// TIA Portal V20 export
FUNCTION_BLOCK "LER_IRCheck_BT5525"   // FB19, LAD
// stored: Access Published, MemoryReserve 100, SetENOAutomatically false
   VAR_INPUT
      enable : Bool;
      enableManualCmds : Bool;
      dryRunCmds : Bool;
   END_VAR
   VAR_OUTPUT
      error : Bool;
      status : Word;
   END_VAR
   VAR_IN_OUT
      controlNode : "LER_typeHipotControlNodes";
      configuration : "LER_typeHipotConfiguration";
      moduleInterface : "LER_typeHipotInterface";
   END_VAR
   VAR
      instSendP2P_type1 { ExternalAccessible := 'False'; ExternalVisible := 'False'; ExternalWritable := 'False'} : Send_P2P;
      instSendP2P_contact { S7_SetPoint := 'True'} : Send_P2P;
      instSendP2P_bddCount { S7_SetPoint := 'True'} : Send_P2P;
      instSendP2P_bddResult { S7_SetPoint := 'True'} : Send_P2P;
      instSendP2P_voltageCmd { S7_SetPoint := 'True'} : Send_P2P;
      instSendP2P_voltageCheck { S7_SetPoint := 'True'} : Send_P2P;
      instSendP2P_timerCmd { S7_SetPoint := 'True'} : Send_P2P;
      instSendP2P_timerCheck { S7_SetPoint := 'True'} : Send_P2P;
      instSendP2P_contactCmd { S7_SetPoint := 'True'} : Send_P2P;
      instSendP2P_contactCheck { S7_SetPoint := 'True'} : Send_P2P;
      instSendP2P_comparatorCmd { S7_SetPoint := 'True'} : Send_P2P;
      instSendP2P_comparatorCheck { S7_SetPoint := 'True'} : Send_P2P;
      instSendP2P_BDD_CCV_cmd { S7_SetPoint := 'True'} : Send_P2P;
      instSendP2P_BDD_CCV_check { S7_SetPoint := 'True'} : Send_P2P;
      instSendP2P_BDD_CVV_cmd { S7_SetPoint := 'True'} : Send_P2P;
      instSendP2P_BDD_CVV_check { S7_SetPoint := 'True'} : Send_P2P;
      instSendP2P_BDD_CVI_cmd { S7_SetPoint := 'True'} : Send_P2P;
      instSendP2P_BDD_CVI_check { S7_SetPoint := 'True'} : Send_P2P;
      instReceiveP2P_type1 { ExternalAccessible := 'False'; ExternalVisible := 'False'; ExternalWritable := 'False'} : Receive_P2P;
      instReceiveP2P_contact { ExternalAccessible := 'False'; ExternalVisible := 'False'; ExternalWritable := 'False'} : Receive_P2P;
      instReceiveP2P_bddCount { ExternalAccessible := 'False'; ExternalVisible := 'False'; ExternalWritable := 'False'} : Receive_P2P;
      instReceiveP2P_bddResult { S7_SetPoint := 'True'} : Receive_P2P;
      instReceiveP2P_voltageCheck { S7_SetPoint := 'True'} : Receive_P2P;
      instReceiveP2P_timerCheck { S7_SetPoint := 'True'} : Receive_P2P;
      instReceiveP2P_contactCheck { S7_SetPoint := 'True'} : Receive_P2P;
      instReceiveP2P_comparatorCheck { S7_SetPoint := 'True'} : Receive_P2P;
      instReceiveP2P_BDD_CCV_check { S7_SetPoint := 'True'} : Receive_P2P;
      instReceiveP2P_BDD_CVV_check { S7_SetPoint := 'True'} : Receive_P2P;
      instReceiveP2P_BDD_CVI_check { S7_SetPoint := 'True'} : Receive_P2P;
      instReceiveReset_type1 { ExternalAccessible := 'False'; ExternalVisible := 'False'; ExternalWritable := 'False'} : Receive_Reset;
      instReceiveReset_contact { S7_SetPoint := 'True'} : Receive_Reset;
      instReceiveReset_bddCount { S7_SetPoint := 'True'} : Receive_Reset;
      instReceiveReset_bddResult { S7_SetPoint := 'True'} : Receive_Reset;
      instReceiveReset_voltageCheck { S7_SetPoint := 'True'} : Receive_Reset;
      instReceiveReset_timerCheck { S7_SetPoint := 'True'} : Receive_Reset;
      instReceiveReset_contactCheck { S7_SetPoint := 'True'} : Receive_Reset;
      instReceiveReset_comparatorCheck { S7_SetPoint := 'True'} : Receive_Reset;
      instReceiveReset_BDD_CCV_check { S7_SetPoint := 'True'} : Receive_Reset;
      instReceiveReset_BDD_CVV_check { S7_SetPoint := 'True'} : Receive_Reset;
      instReceiveReset_BDD_CVI_check { S7_SetPoint := 'True'} : Receive_Reset;
      LER_IRCheck_Calculate_Voltage { S7_SetPoint := 'True'} : "LER_IRCheck_Calculate";
      LER_IRCheck_Calculate_Timer { S7_SetPoint := 'True'} : "LER_IRCheck_Calculate";
      LER_IRCheck_Calculate_ContactCheckLimit { S7_SetPoint := 'True'} : "LER_IRCheck_Calculate";
      LER_IRCheck_Calculate_CompUpperLimit { S7_SetPoint := 'True'} : "LER_IRCheck_Calculate";
      LER_IRCheck_Calculate_CompLowerLimit { S7_SetPoint := 'True'} : "LER_IRCheck_Calculate";
      LER_IRCheck_Calculate_CompLowerLimit_1 { S7_SetPoint := 'True'} : "LER_IRCheck_Calculate";
      LER_IRCheck_Calculate_CompLowerLimit_2 { S7_SetPoint := 'True'} : "LER_IRCheck_Calculate";
      LER_IRCheck_Calculate_CompLowerLimit_3 { S7_SetPoint := 'True'} : "LER_IRCheck_Calculate";
      LER_IRCheck_Calculate_CompLowerLimit_4 { S7_SetPoint := 'True'} : "LER_IRCheck_Calculate";
      LER_IRCheck_Calculate_CompLowerLimit_5 { S7_SetPoint := 'True'} : "LER_IRCheck_Calculate";
      LER_IRCheck_Calculate_BDD_CCV_Set { S7_SetPoint := 'True'} : "LER_IRCheck_Calculate";
      LER_IRCheck_Calculate_BDD_CVV_Set { S7_SetPoint := 'True'} : "LER_IRCheck_Calculate";
      LER_IRCheck_Calculate_BDD_CVI_Set { S7_SetPoint := 'True'} : "LER_IRCheck_Calculate";
      instTON_type1 { S7_SetPoint := 'True'} : Array[0..4] of TON_TIME;
      instTON_contact { S7_SetPoint := 'True'} : Array[0..4] of TON_TIME;
      instTON_bddCount { S7_SetPoint := 'True'} : Array[0..4] of TON_TIME;
      instTON_bddResult { S7_SetPoint := 'True'} : Array[0..4] of TON_TIME;
      instTON_voltage { S7_SetPoint := 'True'} : Array[0..4] of TON_TIME;
      instTON_delayTest { S7_SetPoint := 'True'} : Array[0..4] of TON_TIME;
      statSendP2PLength_type1 { ExternalAccessible := 'False'; ExternalVisible := 'False'; ExternalWritable := 'False'} : UInt;
      statSendP2PLength_contact { ExternalAccessible := 'False'; ExternalVisible := 'False'; ExternalWritable := 'False'} : UInt;
      statSendP2PLength_bddCount { ExternalAccessible := 'False'; ExternalVisible := 'False'; ExternalWritable := 'False'} : UInt;
      statSendP2PLength_bddResult { ExternalAccessible := 'False'; ExternalVisible := 'False'; ExternalWritable := 'False'} : UInt;
      statSendP2PLength_voltageCmd : UInt;
      statSendP2PLength_voltageCheck : UInt;
      statSendP2PLength_timerCmd : UInt;
      statSendP2PLength_timerCheck : UInt;
      statSendP2PLength_contactCmd : UInt;
      statSendP2PLength_contactCheck : UInt;
      statSendP2PLength_comparatorCmd : UInt;
      statSendP2PLength_comparatorCheck : UInt;
      statSendP2PLength_BDD_CCV_cmd : UInt;
      statSendP2PLength_BDD_CCV_check : UInt;
      statSendP2PLength_BDD_CVV_cmd : UInt;
      statSendP2PLength_BDD_CVV_check : UInt;
      statSendP2PLength_BDD_CVI_cmd : UInt;
      statSendP2PLength_BDD_CVI_check : UInt;
      statSendReq_type1 : Bool;
      statSendReq_contact : Bool;
      statSendReq_bddCount : Bool;
      statSendReq_bddResult : Bool;
      statBit_type1 : Array[0..9] of Bool;
      statBit_contact : Array[0..9] of Bool;
      statBit_bddCount : Array[0..9] of Bool;
      statBit_bddResult : Array[0..9] of Bool;
      statSendRequest : Array[0..9999] of Bool;
      statComplete_type1 : Bool;
      statComplete_contact : Bool;
      statComplete_bddCount : Bool;
      statComplete_bddResult : Bool;
      statDataBuffer : Struct
         send_type1 { ExternalAccessible := 'False'; ExternalVisible := 'False'; ExternalWritable := 'False'} : Array[0..49] of Byte;
         rcv_type1 { ExternalAccessible := 'False'; ExternalVisible := 'False'; ExternalWritable := 'False'} : Array[0..49] of Char;
         send_contact { ExternalAccessible := 'False'; ExternalVisible := 'False'; ExternalWritable := 'False'} : Array[0..49] of Byte;
         rcv_contact { ExternalAccessible := 'False'; ExternalVisible := 'False'; ExternalWritable := 'False'} : Array[0..49] of Char;
         send_bddCount { ExternalAccessible := 'False'; ExternalVisible := 'False'; ExternalWritable := 'False'} : Array[0..49] of Byte;
         rcv_bddCount { ExternalAccessible := 'False'; ExternalVisible := 'False'; ExternalWritable := 'False'} : Array[0..49] of Char;
         send_bddResult : Array[0..49] of Byte;
         rcv_bddResult : Array[0..999] of Char;
         send_voltageCmd { ExternalAccessible := 'False'; ExternalVisible := 'False'; ExternalWritable := 'False'} : Array[0..99] of Byte;
         send_voltageCheck { ExternalAccessible := 'False'; ExternalVisible := 'False'; ExternalWritable := 'False'} : Array[0..99] of Byte;
         rcv_voltageCheck : Array[0..99] of Char;
         send_timerCmd { ExternalAccessible := 'False'; ExternalVisible := 'False'; ExternalWritable := 'False'} : Array[0..99] of Byte;
         send_timerCheck { ExternalAccessible := 'False'; ExternalVisible := 'False'; ExternalWritable := 'False'} : Array[0..99] of Byte;
         rcv_timerCheck : Array[0..99] of Char;
         send_contactCmd { ExternalAccessible := 'False'; ExternalVisible := 'False'; ExternalWritable := 'False'} : Array[0..99] of Byte;
         send_contactCheck { ExternalAccessible := 'False'; ExternalVisible := 'False'; ExternalWritable := 'False'} : Array[0..99] of Byte;
         rcv_contactCheck { ExternalAccessible := 'False'; ExternalVisible := 'False'; ExternalWritable := 'False'} : Array[0..99] of Char;
         send_comparatorCmd { ExternalAccessible := 'False'; ExternalVisible := 'False'; ExternalWritable := 'False'} : Array[0..99] of Byte;
         send_comparatorCheck { ExternalAccessible := 'False'; ExternalVisible := 'False'; ExternalWritable := 'False'} : Array[0..99] of Byte;
         rcv_comparatorCheck { ExternalAccessible := 'False'; ExternalVisible := 'False'; ExternalWritable := 'False'} : Array[0..99] of Char;
         send_BDD_CCV_cmd { ExternalAccessible := 'False'; ExternalVisible := 'False'; ExternalWritable := 'False'} : Array[0..99] of Byte;
         send_BDD_CCV_check { ExternalAccessible := 'False'; ExternalVisible := 'False'; ExternalWritable := 'False'} : Array[0..99] of Byte;
         rcv_BDD_CCV_check { ExternalAccessible := 'False'; ExternalVisible := 'False'; ExternalWritable := 'False'} : Array[0..99] of Char;
         send_BDD_CVV_cmd { ExternalAccessible := 'False'; ExternalVisible := 'False'; ExternalWritable := 'False'} : Array[0..99] of Byte;
         send_BDD_CVV_check { ExternalAccessible := 'False'; ExternalVisible := 'False'; ExternalWritable := 'False'} : Array[0..99] of Byte;
         rcv_BDD_CVV_check { ExternalAccessible := 'False'; ExternalVisible := 'False'; ExternalWritable := 'False'} : Array[0..99] of Char;
         send_BDD_CVI_cmd { ExternalAccessible := 'False'; ExternalVisible := 'False'; ExternalWritable := 'False'} : Array[0..99] of Byte;
         send_BDD_CVI_check { ExternalAccessible := 'False'; ExternalVisible := 'False'; ExternalWritable := 'False'} : Array[0..99] of Byte;
         rcv_BDD_CVI_check { ExternalAccessible := 'False'; ExternalVisible := 'False'; ExternalWritable := 'False'} : Array[0..99] of Char;
      END_STRUCT;
      statTrigger : Array[0..9999] of Bool;
      statDataDelete_bddResult { S7_SetPoint := 'True'} : "LER_typeHipotBddData";
      statMonitoring { ExternalAccessible := 'False'; ExternalVisible := 'False'; ExternalWritable := 'False'} : "LER_typeHipotMonitoring";
      statvoltage { S7_SetPoint := 'True'} : String;
      stattimer { S7_SetPoint := 'True'} : String;
      statcompUpperLimit { S7_SetPoint := 'True'} : String;
      statcompLowerLimit { S7_SetPoint := 'True'} : String;
      statcontactCheckLimit { S7_SetPoint := 'True'} : String;
      statBDD_CCV_Set { S7_SetPoint := 'True'} : String;
      statBDD_CVV_Set { S7_SetPoint := 'True'} : String;
      statBDD_CVI_Set { S7_SetPoint := 'True'} : String;
      statStep { ExternalAccessible := 'False'; ExternalVisible := 'False'; ExternalWritable := 'False'} : Int;
      statResultData { ExternalAccessible := 'False'; ExternalVisible := 'False'; ExternalWritable := 'False'} : String[50];
      statRowData_ohm3 { ExternalAccessible := 'False'; ExternalVisible := 'False'; ExternalWritable := 'False'} : String[6];
      statRowData_ohm2 { ExternalAccessible := 'False'; ExternalVisible := 'False'; ExternalWritable := 'False'} : String[3] := ' . ';
      statRowData_ohm1 : String[9];
      statRowData_ohm10 { ExternalAccessible := 'False'; ExternalVisible := 'False'; ExternalWritable := 'False'} : String[5];
      statDword : DWord;
      statHold : Bool;
      statCnt : Array[0..2999] of UInt;
      statTonTimer : Array[0..2999] of TON_TIME;
   END_VAR
   VAR_TEMP
      tempIndex : Int;
      tempBddStringData : String[10];
   END_VAR
   VAR CONSTANT
      delayTime : Time := T#500ms;
      voltageSet : String := ':VOLTage ';
      timerSet : String := ':TIMer ';
      compLimit : String := ':COMParator:';
      contactLimit : String := ':CONTactcheck:CAPacitance:THReshold';
      BDD_CCV_Limit : String := ':BDD:CC:V:THReshold';
      BDD_CVV_Limit : String := ':BDD:CV:V:THReshold';
      BDD_CVI_Limit : String := ':BDD:CV:I:THReshold';
      MOhm_1 : String := 'E6,';
      MOhm_2 : String := 'E6';
      nF : String := 'E-9';
      end : String := 'CRLF';   // < : CR : 16#0D, > : LF : 16#0A
   END_VAR
   // // statMonitoring.result : 1: OK, 2: UFail, 3:LFail, 4:H.ERR, 5:O.F., 6:U.F., 7:C.ERR, 8:Error, 9:INVAL, 10:NOCOMP
   VAR_TEMP   // added for the SCL form of the ladder/FBD networks
      _w1 : Bool;
      _w2 : Bool;
      _w3 : Bool;
      _w4 : Bool;
      _w5 : Bool;
      _w6 : Bool;
      _w7 : Bool;
      _w8 : Bool;
   END_VAR
BEGIN

REGION Network 2: =========================================== Function
END_REGION

REGION Network 3: Type1 send, rcv p2p
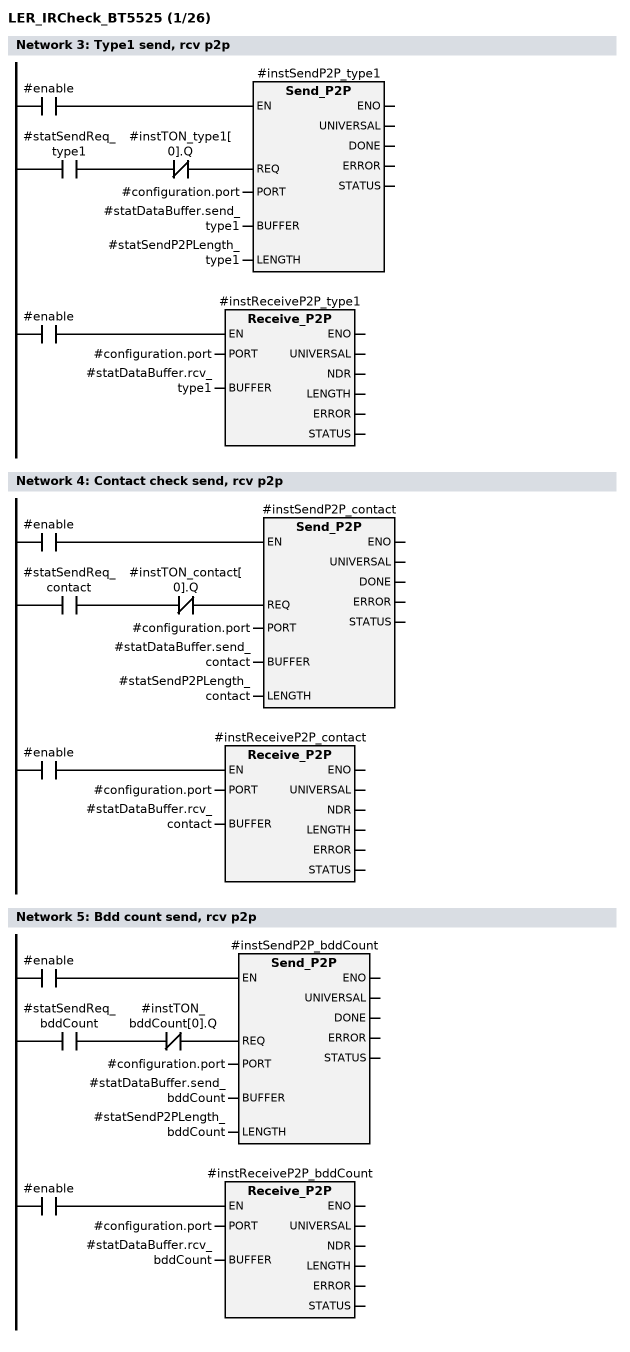
   RUNG wire#powerrail
      Contact( #enable )
      #instSendP2P_type1.Send_P2P(REQ := wire#w1, PORT := #configuration.port, BUFFER := #statDataBuffer.send_type1, LENGTH := #statSendP2PLength_type1, UNIVERSAL =>, DONE =>, ERROR =>, STATUS =>)
   END_RUNG
   RUNG wire#powerrail
      Contact( #statSendReq_type1 )
      I_Contact( #instTON_type1[0].Q )
   END_RUNG wire#w1
   RUNG wire#powerrail
      Contact( #enable )
      #instReceiveP2P_type1.Receive_P2P(PORT := #configuration.port, BUFFER := #statDataBuffer.rcv_type1, UNIVERSAL =>, NDR =>, LENGTH =>, ERROR =>, STATUS =>)
   END_RUNG
   // the same network as SCL:
   IF #enable THEN
       #instSendP2P_type1(REQ := #statSendReq_type1 AND NOT #instTON_type1[0].Q,   // Send_P2P
                          PORT := #configuration.port,
                          BUFFER := #statDataBuffer.send_type1,
                          LENGTH := #statSendP2PLength_type1);
       #instReceiveP2P_type1(PORT := #configuration.port, BUFFER := #statDataBuffer.rcv_type1);   // Receive_P2P
   END_IF;
END_REGION

REGION Network 4: Contact check send, rcv p2p
   RUNG wire#powerrail
      Contact( #enable )
      #instSendP2P_contact.Send_P2P(REQ := wire#w1, PORT := #configuration.port, BUFFER := #statDataBuffer.send_contact, LENGTH := #statSendP2PLength_contact, UNIVERSAL =>, DONE =>, ERROR =>, STATUS =>)
   END_RUNG
   RUNG wire#powerrail
      Contact( #statSendReq_contact )
      I_Contact( #instTON_contact[0].Q )
   END_RUNG wire#w1
   RUNG wire#powerrail
      Contact( #enable )
      #instReceiveP2P_contact.Receive_P2P(PORT := #configuration.port, BUFFER := #statDataBuffer.rcv_contact, UNIVERSAL =>, NDR =>, LENGTH =>, ERROR =>, STATUS =>)
   END_RUNG
   // the same network as SCL:
   IF #enable THEN
       #instSendP2P_contact(REQ := #statSendReq_contact AND NOT #instTON_contact[0].Q,   // Send_P2P
                            PORT := #configuration.port,
                            BUFFER := #statDataBuffer.send_contact,
                            LENGTH := #statSendP2PLength_contact);
       #instReceiveP2P_contact(PORT := #configuration.port, BUFFER := #statDataBuffer.rcv_contact);   // Receive_P2P
   END_IF;
END_REGION

REGION Network 5: Bdd count send, rcv p2p
   RUNG wire#powerrail
      Contact( #enable )
      #instSendP2P_bddCount.Send_P2P(REQ := wire#w1, PORT := #configuration.port, BUFFER := #statDataBuffer.send_bddCount, LENGTH := #statSendP2PLength_bddCount, UNIVERSAL =>, DONE =>, ERROR =>, STATUS =>)
   END_RUNG
   RUNG wire#powerrail
      Contact( #statSendReq_bddCount )
      I_Contact( #instTON_bddCount[0].Q )
   END_RUNG wire#w1
   RUNG wire#powerrail
      Contact( #enable )
      #instReceiveP2P_bddCount.Receive_P2P(PORT := #configuration.port, BUFFER := #statDataBuffer.rcv_bddCount, UNIVERSAL =>, NDR =>, LENGTH =>, ERROR =>, STATUS =>)
   END_RUNG
   // the same network as SCL:
   IF #enable THEN
       #instSendP2P_bddCount(REQ := #statSendReq_bddCount AND NOT #instTON_bddCount[0].Q,   // Send_P2P
                             PORT := #configuration.port,
                             BUFFER := #statDataBuffer.send_bddCount,
                             LENGTH := #statSendP2PLength_bddCount);
       #instReceiveP2P_bddCount(PORT := #configuration.port, BUFFER := #statDataBuffer.rcv_bddCount);   // Receive_P2P
   END_IF;
END_REGION

REGION Network 6: Bdd result send, rcv p2p
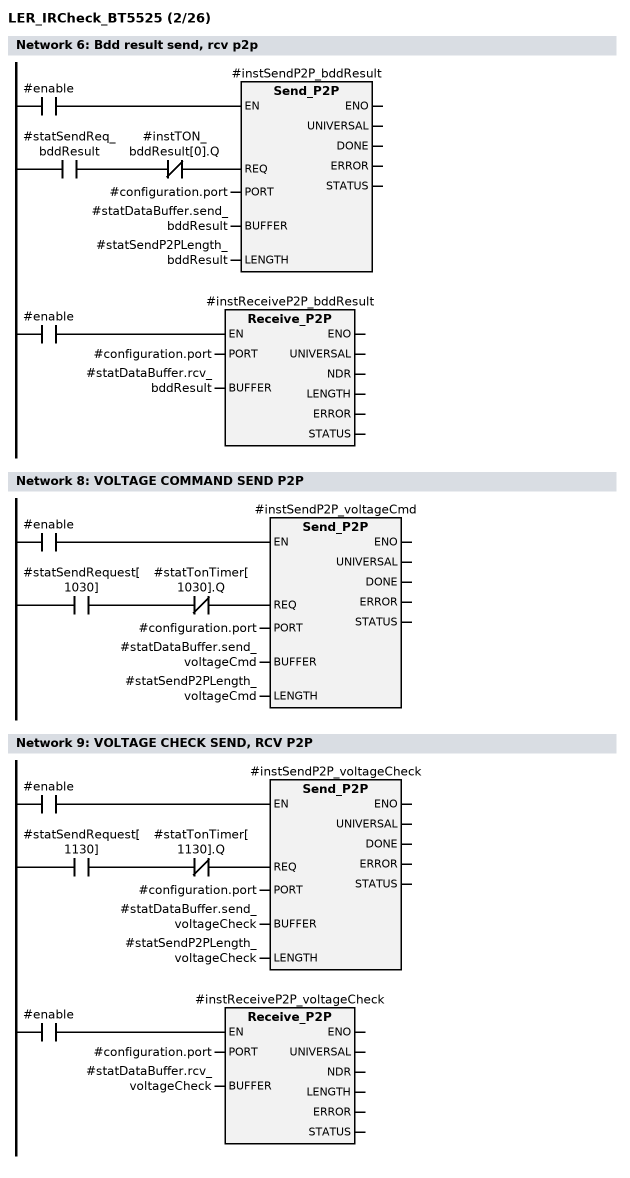
   RUNG wire#powerrail
      Contact( #enable )
      #instSendP2P_bddResult.Send_P2P(REQ := wire#w1, PORT := #configuration.port, BUFFER := #statDataBuffer.send_bddResult, LENGTH := #statSendP2PLength_bddResult, UNIVERSAL =>, DONE =>, ERROR =>, STATUS =>)
   END_RUNG
   RUNG wire#powerrail
      Contact( #statSendReq_bddResult )
      I_Contact( #instTON_bddResult[0].Q )
   END_RUNG wire#w1
   RUNG wire#powerrail
      Contact( #enable )
      #instReceiveP2P_bddResult.Receive_P2P(PORT := #configuration.port, BUFFER := #statDataBuffer.rcv_bddResult, UNIVERSAL =>, NDR =>, LENGTH =>, ERROR =>, STATUS =>)
   END_RUNG
   // the same network as SCL:
   IF #enable THEN
       #instSendP2P_bddResult(REQ := #statSendReq_bddResult AND NOT #instTON_bddResult[0].Q,   // Send_P2P
                              PORT := #configuration.port,
                              BUFFER := #statDataBuffer.send_bddResult,
                              LENGTH := #statSendP2PLength_bddResult);
       #instReceiveP2P_bddResult(PORT := #configuration.port, BUFFER := #statDataBuffer.rcv_bddResult);   // Receive_P2P
   END_IF;
END_REGION

REGION Network 7: =========================================== FUNCTION [PARAMETER]
END_REGION

REGION Network 8: VOLTAGE COMMAND SEND P2P
   RUNG wire#powerrail
      Contact( #enable )
      #instSendP2P_voltageCmd.Send_P2P(REQ := wire#w1, PORT := #configuration.port, BUFFER := #statDataBuffer.send_voltageCmd, LENGTH := #statSendP2PLength_voltageCmd, UNIVERSAL =>, DONE =>, ERROR =>, STATUS =>)
   END_RUNG
   RUNG wire#powerrail
      Contact( #statSendRequest[1030] )
      I_Contact( #statTonTimer[1030].Q )
   END_RUNG wire#w1
   // the same network as SCL:
   IF #enable THEN
       #instSendP2P_voltageCmd(REQ := #statSendRequest[1030] AND NOT #statTonTimer[1030].Q,   // Send_P2P
                               PORT := #configuration.port,
                               BUFFER := #statDataBuffer.send_voltageCmd,
                               LENGTH := #statSendP2PLength_voltageCmd);
   END_IF;
END_REGION

REGION Network 9: VOLTAGE CHECK SEND, RCV P2P
   RUNG wire#powerrail
      Contact( #enable )
      #instSendP2P_voltageCheck.Send_P2P(REQ := wire#w1, PORT := #configuration.port, BUFFER := #statDataBuffer.send_voltageCheck, LENGTH := #statSendP2PLength_voltageCheck, UNIVERSAL =>, DONE =>, ERROR =>, STATUS =>)
   END_RUNG
   RUNG wire#powerrail
      Contact( #statSendRequest[1130] )
      I_Contact( #statTonTimer[1130].Q )
   END_RUNG wire#w1
   RUNG wire#powerrail
      Contact( #enable )
      #instReceiveP2P_voltageCheck.Receive_P2P(PORT := #configuration.port, BUFFER := #statDataBuffer.rcv_voltageCheck, UNIVERSAL =>, NDR =>, LENGTH =>, ERROR =>, STATUS =>)
   END_RUNG
   // the same network as SCL:
   IF #enable THEN
       #instSendP2P_voltageCheck(REQ := #statSendRequest[1130] AND NOT #statTonTimer[1130].Q,   // Send_P2P
                               PORT := #configuration.port,
                               BUFFER := #statDataBuffer.send_voltageCheck,
                               LENGTH := #statSendP2PLength_voltageCheck);
       #instReceiveP2P_voltageCheck(PORT := #configuration.port, BUFFER := #statDataBuffer.rcv_voltageCheck);   // Receive_P2P
   END_IF;
END_REGION

REGION Network 10: TIMER COMMAND SEND P2P
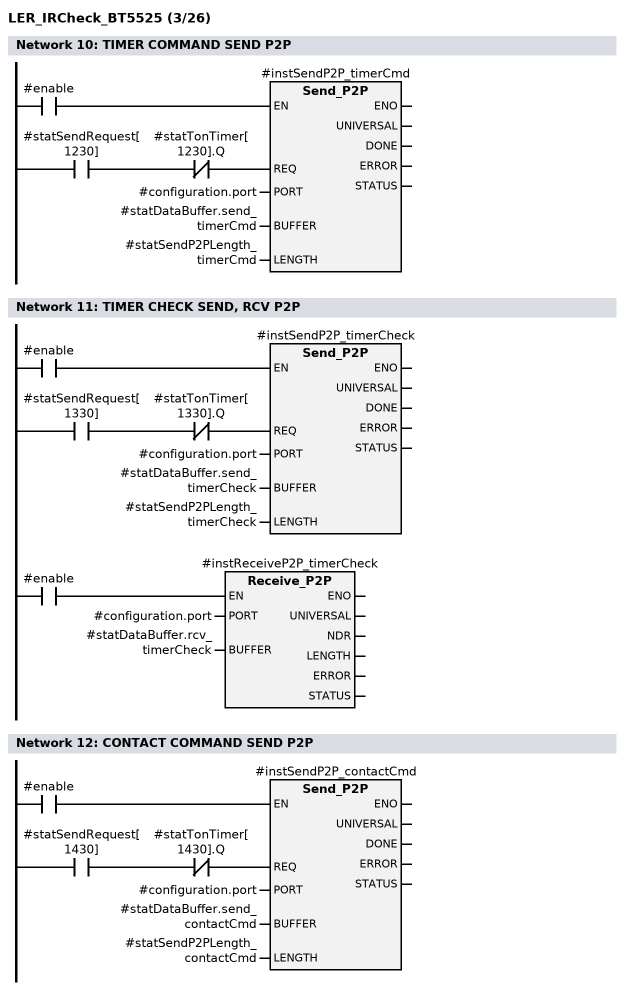
   RUNG wire#powerrail
      Contact( #enable )
      #instSendP2P_timerCmd.Send_P2P(REQ := wire#w1, PORT := #configuration.port, BUFFER := #statDataBuffer.send_timerCmd, LENGTH := #statSendP2PLength_timerCmd, UNIVERSAL =>, DONE =>, ERROR =>, STATUS =>)
   END_RUNG
   RUNG wire#powerrail
      Contact( #statSendRequest[1230] )
      I_Contact( #statTonTimer[1230].Q )
   END_RUNG wire#w1
   // the same network as SCL:
   IF #enable THEN
       #instSendP2P_timerCmd(REQ := #statSendRequest[1230] AND NOT #statTonTimer[1230].Q,   // Send_P2P
                             PORT := #configuration.port,
                             BUFFER := #statDataBuffer.send_timerCmd,
                             LENGTH := #statSendP2PLength_timerCmd);
   END_IF;
END_REGION

REGION Network 11: TIMER CHECK SEND, RCV P2P
   RUNG wire#powerrail
      Contact( #enable )
      #instSendP2P_timerCheck.Send_P2P(REQ := wire#w1, PORT := #configuration.port, BUFFER := #statDataBuffer.send_timerCheck, LENGTH := #statSendP2PLength_timerCheck, UNIVERSAL =>, DONE =>, ERROR =>, STATUS =>)
   END_RUNG
   RUNG wire#powerrail
      Contact( #statSendRequest[1330] )
      I_Contact( #statTonTimer[1330].Q )
   END_RUNG wire#w1
   RUNG wire#powerrail
      Contact( #enable )
      #instReceiveP2P_timerCheck.Receive_P2P(PORT := #configuration.port, BUFFER := #statDataBuffer.rcv_timerCheck, UNIVERSAL =>, NDR =>, LENGTH =>, ERROR =>, STATUS =>)
   END_RUNG
   // the same network as SCL:
   IF #enable THEN
       #instSendP2P_timerCheck(REQ := #statSendRequest[1330] AND NOT #statTonTimer[1330].Q,   // Send_P2P
                               PORT := #configuration.port,
                               BUFFER := #statDataBuffer.send_timerCheck,
                               LENGTH := #statSendP2PLength_timerCheck);
       #instReceiveP2P_timerCheck(PORT := #configuration.port, BUFFER := #statDataBuffer.rcv_timerCheck);   // Receive_P2P
   END_IF;
END_REGION

REGION Network 12: CONTACT COMMAND SEND P2P
   RUNG wire#powerrail
      Contact( #enable )
      #instSendP2P_contactCmd.Send_P2P(REQ := wire#w1, PORT := #configuration.port, BUFFER := #statDataBuffer.send_contactCmd, LENGTH := #statSendP2PLength_contactCmd, UNIVERSAL =>, DONE =>, ERROR =>, STATUS =>)
   END_RUNG
   RUNG wire#powerrail
      Contact( #statSendRequest[1430] )
      I_Contact( #statTonTimer[1430].Q )
   END_RUNG wire#w1
   // the same network as SCL:
   IF #enable THEN
       #instSendP2P_contactCmd(REQ := #statSendRequest[1430] AND NOT #statTonTimer[1430].Q,   // Send_P2P
                               PORT := #configuration.port,
                               BUFFER := #statDataBuffer.send_contactCmd,
                               LENGTH := #statSendP2PLength_contactCmd);
   END_IF;
END_REGION

REGION Network 13: CONTACT CHECK SEND, RCV P2P
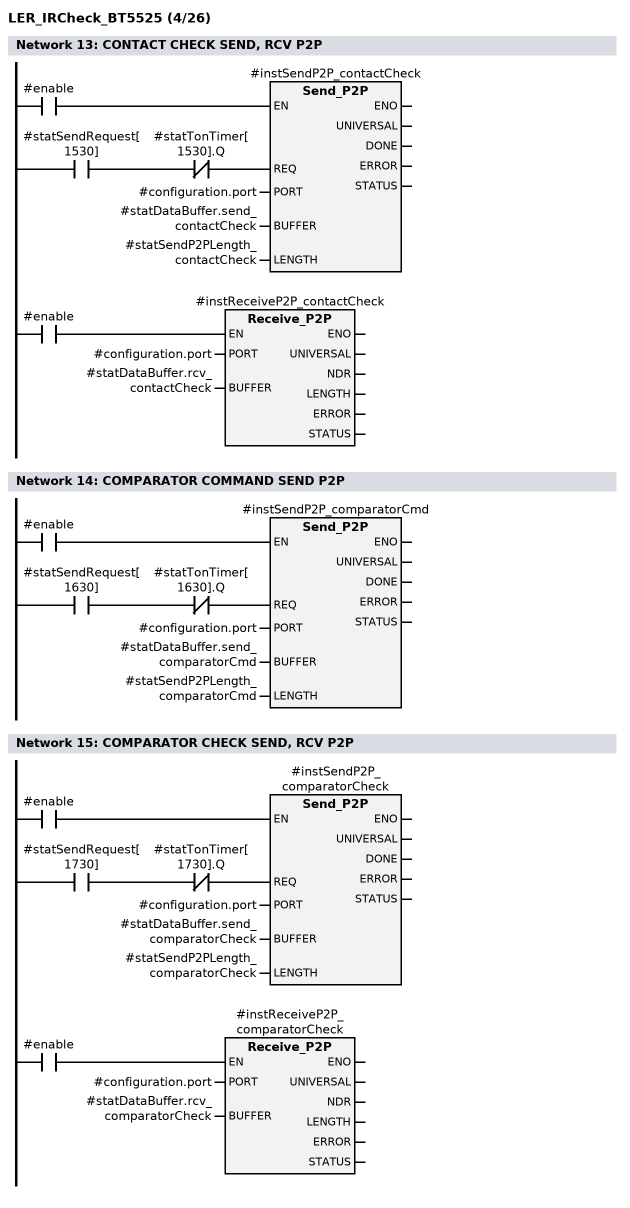
   RUNG wire#powerrail
      Contact( #enable )
      #instSendP2P_contactCheck.Send_P2P(REQ := wire#w1, PORT := #configuration.port, BUFFER := #statDataBuffer.send_contactCheck, LENGTH := #statSendP2PLength_contactCheck, UNIVERSAL =>, DONE =>, ERROR =>, STATUS =>)
   END_RUNG
   RUNG wire#powerrail
      Contact( #statSendRequest[1530] )
      I_Contact( #statTonTimer[1530].Q )
   END_RUNG wire#w1
   RUNG wire#powerrail
      Contact( #enable )
      #instReceiveP2P_contactCheck.Receive_P2P(PORT := #configuration.port, BUFFER := #statDataBuffer.rcv_contactCheck, UNIVERSAL =>, NDR =>, LENGTH =>, ERROR =>, STATUS =>)
   END_RUNG
   // the same network as SCL:
   IF #enable THEN
       #instSendP2P_contactCheck(REQ := #statSendRequest[1530] AND NOT #statTonTimer[1530].Q,   // Send_P2P
                               PORT := #configuration.port,
                               BUFFER := #statDataBuffer.send_contactCheck,
                               LENGTH := #statSendP2PLength_contactCheck);
       #instReceiveP2P_contactCheck(PORT := #configuration.port, BUFFER := #statDataBuffer.rcv_contactCheck);   // Receive_P2P
   END_IF;
END_REGION

REGION Network 14: COMPARATOR COMMAND SEND P2P
   RUNG wire#powerrail
      Contact( #enable )
      #instSendP2P_comparatorCmd.Send_P2P(REQ := wire#w1, PORT := #configuration.port, BUFFER := #statDataBuffer.send_comparatorCmd, LENGTH := #statSendP2PLength_comparatorCmd, UNIVERSAL =>, DONE =>, ERROR =>, STATUS =>)
   END_RUNG
   RUNG wire#powerrail
      Contact( #statSendRequest[1630] )
      I_Contact( #statTonTimer[1630].Q )
   END_RUNG wire#w1
   // the same network as SCL:
   IF #enable THEN
       #instSendP2P_comparatorCmd(REQ := #statSendRequest[1630] AND NOT #statTonTimer[1630].Q,   // Send_P2P
                               PORT := #configuration.port,
                               BUFFER := #statDataBuffer.send_comparatorCmd,
                               LENGTH := #statSendP2PLength_comparatorCmd);
   END_IF;
END_REGION

REGION Network 15: COMPARATOR CHECK SEND, RCV P2P
   RUNG wire#powerrail
      Contact( #enable )
      #instSendP2P_comparatorCheck.Send_P2P(REQ := wire#w1, PORT := #configuration.port, BUFFER := #statDataBuffer.send_comparatorCheck, LENGTH := #statSendP2PLength_comparatorCheck, UNIVERSAL =>, DONE =>, ERROR =>, STATUS =>)
   END_RUNG
   RUNG wire#powerrail
      Contact( #statSendRequest[1730] )
      I_Contact( #statTonTimer[1730].Q )
   END_RUNG wire#w1
   RUNG wire#powerrail
      Contact( #enable )
      #instReceiveP2P_comparatorCheck.Receive_P2P(PORT := #configuration.port, BUFFER := #statDataBuffer.rcv_comparatorCheck, UNIVERSAL =>, NDR =>, LENGTH =>, ERROR =>, STATUS =>)
   END_RUNG
   // the same network as SCL:
   IF #enable THEN
       #instSendP2P_comparatorCheck(REQ := #statSendRequest[1730] AND NOT #statTonTimer[1730].Q,   // Send_P2P
                               PORT := #configuration.port,
                               BUFFER := #statDataBuffer.send_comparatorCheck,
                               LENGTH := #statSendP2PLength_comparatorCheck);
       #instReceiveP2P_comparatorCheck(PORT := #configuration.port, BUFFER := #statDataBuffer.rcv_comparatorCheck);   // Receive_P2P
   END_IF;
END_REGION

REGION Network 16: BDD CCV COMMAND SEND P2P
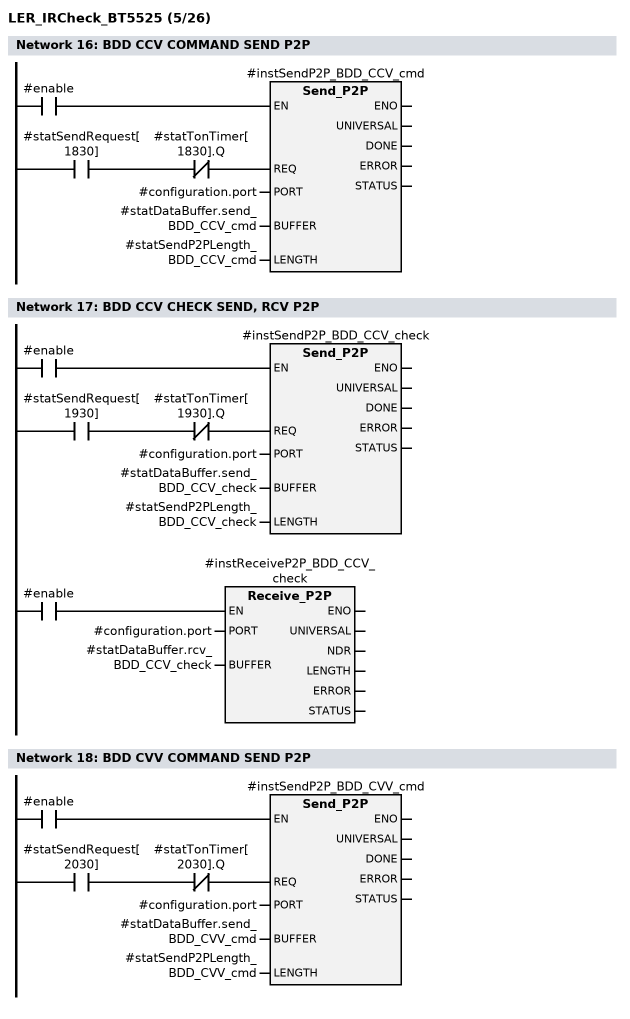
   RUNG wire#powerrail
      Contact( #enable )
      #instSendP2P_BDD_CCV_cmd.Send_P2P(REQ := wire#w1, PORT := #configuration.port, BUFFER := #statDataBuffer.send_BDD_CCV_cmd, LENGTH := #statSendP2PLength_BDD_CCV_cmd, UNIVERSAL =>, DONE =>, ERROR =>, STATUS =>)
   END_RUNG
   RUNG wire#powerrail
      Contact( #statSendRequest[1830] )
      I_Contact( #statTonTimer[1830].Q )
   END_RUNG wire#w1
   // the same network as SCL:
   IF #enable THEN
       #instSendP2P_BDD_CCV_cmd(REQ := #statSendRequest[1830] AND NOT #statTonTimer[1830].Q,   // Send_P2P
                               PORT := #configuration.port,
                               BUFFER := #statDataBuffer.send_BDD_CCV_cmd,
                               LENGTH := #statSendP2PLength_BDD_CCV_cmd);
   END_IF;
END_REGION

REGION Network 17: BDD CCV CHECK SEND, RCV P2P
   RUNG wire#powerrail
      Contact( #enable )
      #instSendP2P_BDD_CCV_check.Send_P2P(REQ := wire#w1, PORT := #configuration.port, BUFFER := #statDataBuffer.send_BDD_CCV_check, LENGTH := #statSendP2PLength_BDD_CCV_check, UNIVERSAL =>, DONE =>, ERROR =>, STATUS =>)
   END_RUNG
   RUNG wire#powerrail
      Contact( #statSendRequest[1930] )
      I_Contact( #statTonTimer[1930].Q )
   END_RUNG wire#w1
   RUNG wire#powerrail
      Contact( #enable )
      #instReceiveP2P_BDD_CCV_check.Receive_P2P(PORT := #configuration.port, BUFFER := #statDataBuffer.rcv_BDD_CCV_check, UNIVERSAL =>, NDR =>, LENGTH =>, ERROR =>, STATUS =>)
   END_RUNG
   // the same network as SCL:
   IF #enable THEN
       #instSendP2P_BDD_CCV_check(REQ := #statSendRequest[1930] AND NOT #statTonTimer[1930].Q,   // Send_P2P
                               PORT := #configuration.port,
                               BUFFER := #statDataBuffer.send_BDD_CCV_check,
                               LENGTH := #statSendP2PLength_BDD_CCV_check);
       #instReceiveP2P_BDD_CCV_check(PORT := #configuration.port, BUFFER := #statDataBuffer.rcv_BDD_CCV_check);   // Receive_P2P
   END_IF;
END_REGION

REGION Network 18: BDD CVV COMMAND SEND P2P
   RUNG wire#powerrail
      Contact( #enable )
      #instSendP2P_BDD_CVV_cmd.Send_P2P(REQ := wire#w1, PORT := #configuration.port, BUFFER := #statDataBuffer.send_BDD_CVV_cmd, LENGTH := #statSendP2PLength_BDD_CVV_cmd, UNIVERSAL =>, DONE =>, ERROR =>, STATUS =>)
   END_RUNG
   RUNG wire#powerrail
      Contact( #statSendRequest[2030] )
      I_Contact( #statTonTimer[2030].Q )
   END_RUNG wire#w1
   // the same network as SCL:
   IF #enable THEN
       #instSendP2P_BDD_CVV_cmd(REQ := #statSendRequest[2030] AND NOT #statTonTimer[2030].Q,   // Send_P2P
                               PORT := #configuration.port,
                               BUFFER := #statDataBuffer.send_BDD_CVV_cmd,
                               LENGTH := #statSendP2PLength_BDD_CVV_cmd);
   END_IF;
END_REGION

REGION Network 19: BDD CVV CHECK SEND, RCV P2P
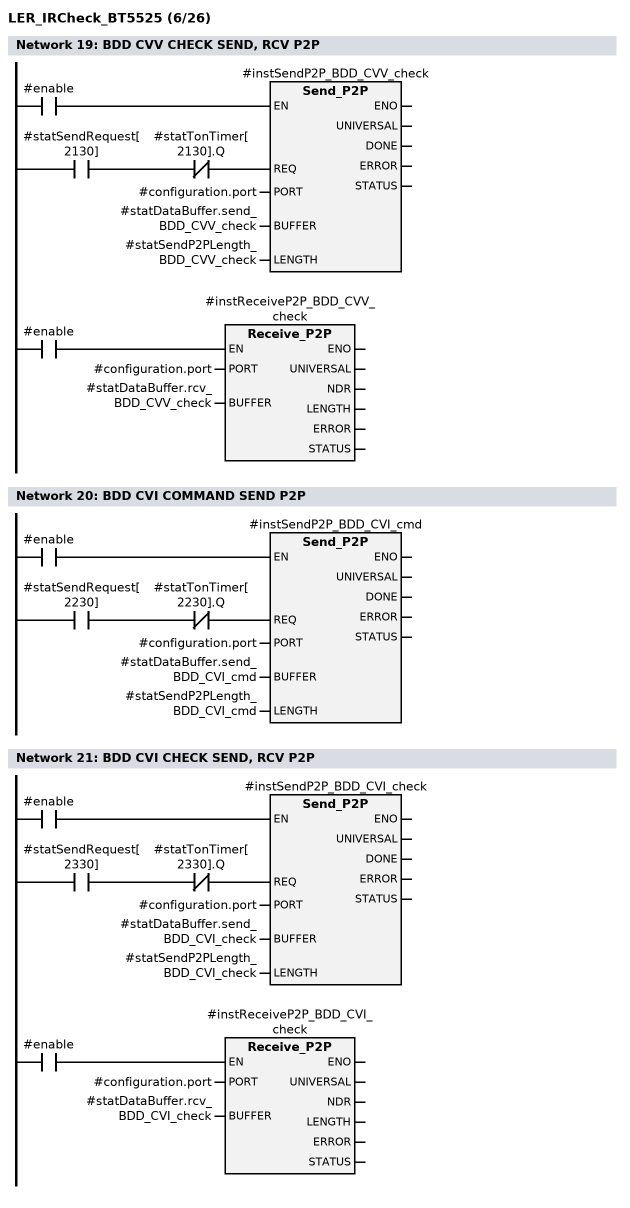
   RUNG wire#powerrail
      Contact( #enable )
      #instSendP2P_BDD_CVV_check.Send_P2P(REQ := wire#w1, PORT := #configuration.port, BUFFER := #statDataBuffer.send_BDD_CVV_check, LENGTH := #statSendP2PLength_BDD_CVV_check, UNIVERSAL =>, DONE =>, ERROR =>, STATUS =>)
   END_RUNG
   RUNG wire#powerrail
      Contact( #statSendRequest[2130] )
      I_Contact( #statTonTimer[2130].Q )
   END_RUNG wire#w1
   RUNG wire#powerrail
      Contact( #enable )
      #instReceiveP2P_BDD_CVV_check.Receive_P2P(PORT := #configuration.port, BUFFER := #statDataBuffer.rcv_BDD_CVV_check, UNIVERSAL =>, NDR =>, LENGTH =>, ERROR =>, STATUS =>)
   END_RUNG
   // the same network as SCL:
   IF #enable THEN
       #instSendP2P_BDD_CVV_check(REQ := #statSendRequest[2130] AND NOT #statTonTimer[2130].Q,   // Send_P2P
                               PORT := #configuration.port,
                               BUFFER := #statDataBuffer.send_BDD_CVV_check,
                               LENGTH := #statSendP2PLength_BDD_CVV_check);
       #instReceiveP2P_BDD_CVV_check(PORT := #configuration.port, BUFFER := #statDataBuffer.rcv_BDD_CVV_check);   // Receive_P2P
   END_IF;
END_REGION

REGION Network 20: BDD CVI COMMAND SEND P2P
   RUNG wire#powerrail
      Contact( #enable )
      #instSendP2P_BDD_CVI_cmd.Send_P2P(REQ := wire#w1, PORT := #configuration.port, BUFFER := #statDataBuffer.send_BDD_CVI_cmd, LENGTH := #statSendP2PLength_BDD_CVI_cmd, UNIVERSAL =>, DONE =>, ERROR =>, STATUS =>)
   END_RUNG
   RUNG wire#powerrail
      Contact( #statSendRequest[2230] )
      I_Contact( #statTonTimer[2230].Q )
   END_RUNG wire#w1
   // the same network as SCL:
   IF #enable THEN
       #instSendP2P_BDD_CVI_cmd(REQ := #statSendRequest[2230] AND NOT #statTonTimer[2230].Q,   // Send_P2P
                               PORT := #configuration.port,
                               BUFFER := #statDataBuffer.send_BDD_CVI_cmd,
                               LENGTH := #statSendP2PLength_BDD_CVI_cmd);
   END_IF;
END_REGION

REGION Network 21: BDD CVI CHECK SEND, RCV P2P
   RUNG wire#powerrail
      Contact( #enable )
      #instSendP2P_BDD_CVI_check.Send_P2P(REQ := wire#w1, PORT := #configuration.port, BUFFER := #statDataBuffer.send_BDD_CVI_check, LENGTH := #statSendP2PLength_BDD_CVI_check, UNIVERSAL =>, DONE =>, ERROR =>, STATUS =>)
   END_RUNG
   RUNG wire#powerrail
      Contact( #statSendRequest[2330] )
      I_Contact( #statTonTimer[2330].Q )
   END_RUNG wire#w1
   RUNG wire#powerrail
      Contact( #enable )
      #instReceiveP2P_BDD_CVI_check.Receive_P2P(PORT := #configuration.port, BUFFER := #statDataBuffer.rcv_BDD_CVI_check, UNIVERSAL =>, NDR =>, LENGTH =>, ERROR =>, STATUS =>)
   END_RUNG
   // the same network as SCL:
   IF #enable THEN
       #instSendP2P_BDD_CVI_check(REQ := #statSendRequest[2330] AND NOT #statTonTimer[2330].Q,   // Send_P2P
                               PORT := #configuration.port,
                               BUFFER := #statDataBuffer.send_BDD_CVI_check,
                               LENGTH := #statSendP2PLength_BDD_CVI_check);
       #instReceiveP2P_BDD_CVI_check(PORT := #configuration.port, BUFFER := #statDataBuffer.rcv_BDD_CVI_check);   // Receive_P2P
   END_IF;
END_REGION

REGION Network 22: =========================================== Mapping
END_REGION

REGION Network 23 (SCL): Input mapping
   REGION Input mapping



   END_REGION
END_REGION

REGION Network 24: =========================================== Sequence step 0 ~
END_REGION

REGION Network 25: STEP 0 : READY
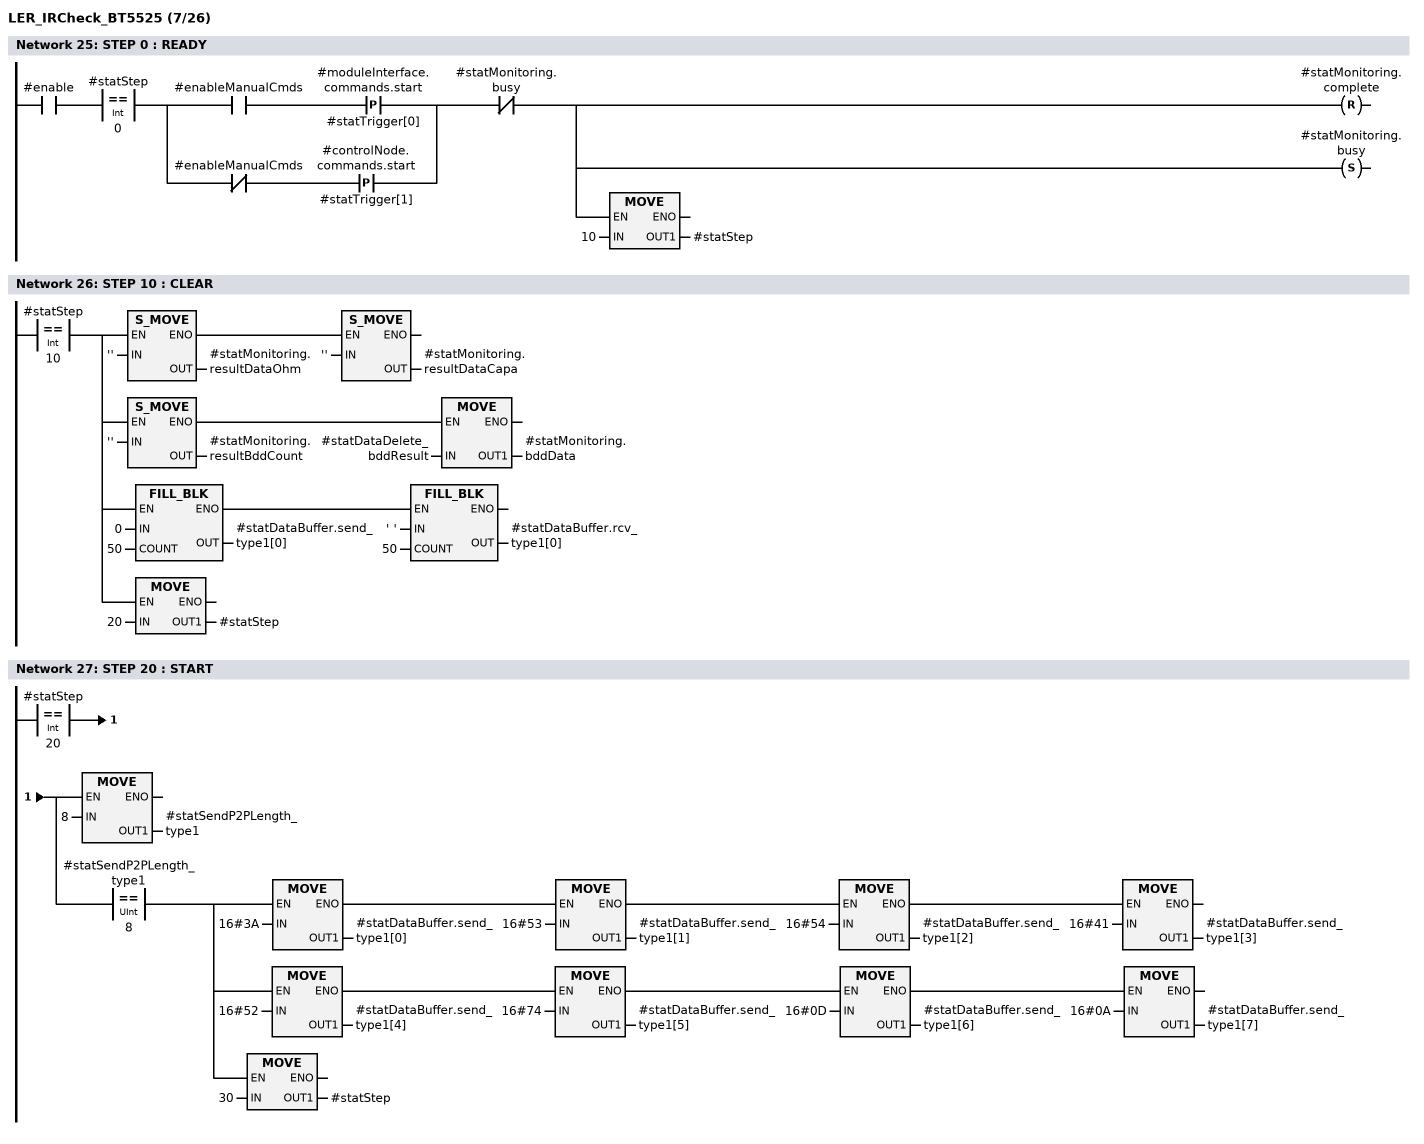
   RUNG wire#powerrail
      Contact( #enable )
      { S7_Templates := "SrcType := Int" } EQ_Contact(in1 := #statStep, in2 := 0)
      wire#w1
      Contact( #enableManualCmds )
      P_Contact(operand := #moduleInterface.commands.start, bit := #statTrigger[0])
      wire#w2
      I_Contact( #statMonitoring.busy )
      wire#w3
      R_Coil( #statMonitoring.complete )
   END_RUNG
   RUNG wire#w1
      I_Contact( #enableManualCmds )
      P_Contact(operand := #controlNode.commands.start, bit := #statTrigger[1])
   END_RUNG wire#w2
   RUNG wire#w3
      S_Coil( #statMonitoring.busy )
   END_RUNG
   RUNG wire#w3
      Move(in := 10, out1 => #statStep)
   END_RUNG
   // the same network as SCL:
   #_w1 := #enable AND (#statStep = 0) AND #enableManualCmds AND #moduleInterface.commands.start AND NOT #statTrigger[0];   // rising edge of #moduleInterface.commands.start
   #statTrigger[0] := #moduleInterface.commands.start;
   #_w2 := #enable AND (#statStep = 0) AND NOT #enableManualCmds AND #controlNode.commands.start AND NOT #statTrigger[1];   // rising edge of #controlNode.commands.start
   #statTrigger[1] := #controlNode.commands.start;
   IF (#_w1 OR #_w2) AND NOT #statMonitoring.busy THEN #statMonitoring.complete := FALSE; END_IF;
   #_w3 := (#_w1 OR #_w2) AND NOT #statMonitoring.busy;
   IF #_w3 THEN
       #statMonitoring.busy := TRUE;
       #statStep := 10;
   END_IF;
END_REGION

REGION Network 26: STEP 10 : CLEAR
   RUNG wire#powerrail
      { S7_Templates := "SrcType := Int" } EQ_Contact(in1 := #statStep, in2 := 10)
      wire#w1
      S_Move(in := '', out => #statMonitoring.resultDataOhm)
      S_Move(in := '', out => #statMonitoring.resultDataCapa)
   END_RUNG
   RUNG wire#w1
      S_Move(in := '', out => #statMonitoring.resultBddCount)
      Move(in := #statDataDelete_bddResult, out1 => #statMonitoring.bddData)
   END_RUNG
   RUNG wire#w1
      FillBlockI(in := 0, count := 50, out => #statDataBuffer.send_type1[0])
      FillBlockI(in := ' ', count := 50, out => #statDataBuffer.rcv_type1[0])
   END_RUNG
   RUNG wire#w1
      Move(in := 20, out1 => #statStep)
   END_RUNG
   // the same network as SCL:
   IF #statStep = 10 THEN
       #statMonitoring.resultDataOhm := '';
       #statMonitoring.resultDataCapa := '';
       #statMonitoring.resultBddCount := '';
       #statMonitoring.bddData := #statDataDelete_bddResult;
       FILL_BLK(IN := 0, COUNT := 50, OUT => #statDataBuffer.send_type1[0]);
       FILL_BLK(IN := ' ', COUNT := 50, OUT => #statDataBuffer.rcv_type1[0]);
       #statStep := 20;
   END_IF;
END_REGION

REGION Network 27: STEP 20 : START
   RUNG wire#powerrail
      { S7_Templates := "SrcType := Int" } EQ_Contact(in1 := #statStep, in2 := 20)
      wire#w1
      Move(in := 8, out1 => #statSendP2PLength_type1)
   END_RUNG
   RUNG wire#w1
      { S7_Templates := "SrcType := UInt" } EQ_Contact(in1 := #statSendP2PLength_type1, in2 := 8)
      wire#w2
      Move(in := 16#3A, out1 => #statDataBuffer.send_type1[0])
      Move(in := 16#53, out1 => #statDataBuffer.send_type1[1])
      Move(in := 16#54, out1 => #statDataBuffer.send_type1[2])
      Move(in := 16#41, out1 => #statDataBuffer.send_type1[3])
   END_RUNG
   RUNG wire#w2
      Move(in := 16#52, out1 => #statDataBuffer.send_type1[4])
      Move(in := 16#74, out1 => #statDataBuffer.send_type1[5])
      Move(in := 16#0D, out1 => #statDataBuffer.send_type1[6])
      Move(in := 16#0A, out1 => #statDataBuffer.send_type1[7])
   END_RUNG
   RUNG wire#w2
      Move(in := 30, out1 => #statStep)
   END_RUNG
   // the same network as SCL:
   #_w1 := #statStep = 20;
   IF #_w1 THEN #statSendP2PLength_type1 := 8; END_IF;
   IF #_w1 AND (#statSendP2PLength_type1 = 8) THEN
       #statDataBuffer.send_type1[0] := 16#3A;
       #statDataBuffer.send_type1[1] := 16#53;
       #statDataBuffer.send_type1[2] := 16#54;
       #statDataBuffer.send_type1[3] := 16#41;
       #statDataBuffer.send_type1[4] := 16#52;
       #statDataBuffer.send_type1[5] := 16#74;
       #statDataBuffer.send_type1[6] := 16#0D;
       #statDataBuffer.send_type1[7] := 16#0A;
       #statStep := 30;
   END_IF;
END_REGION

REGION Network 28: STEP 30 : SEND P2P REQUEST
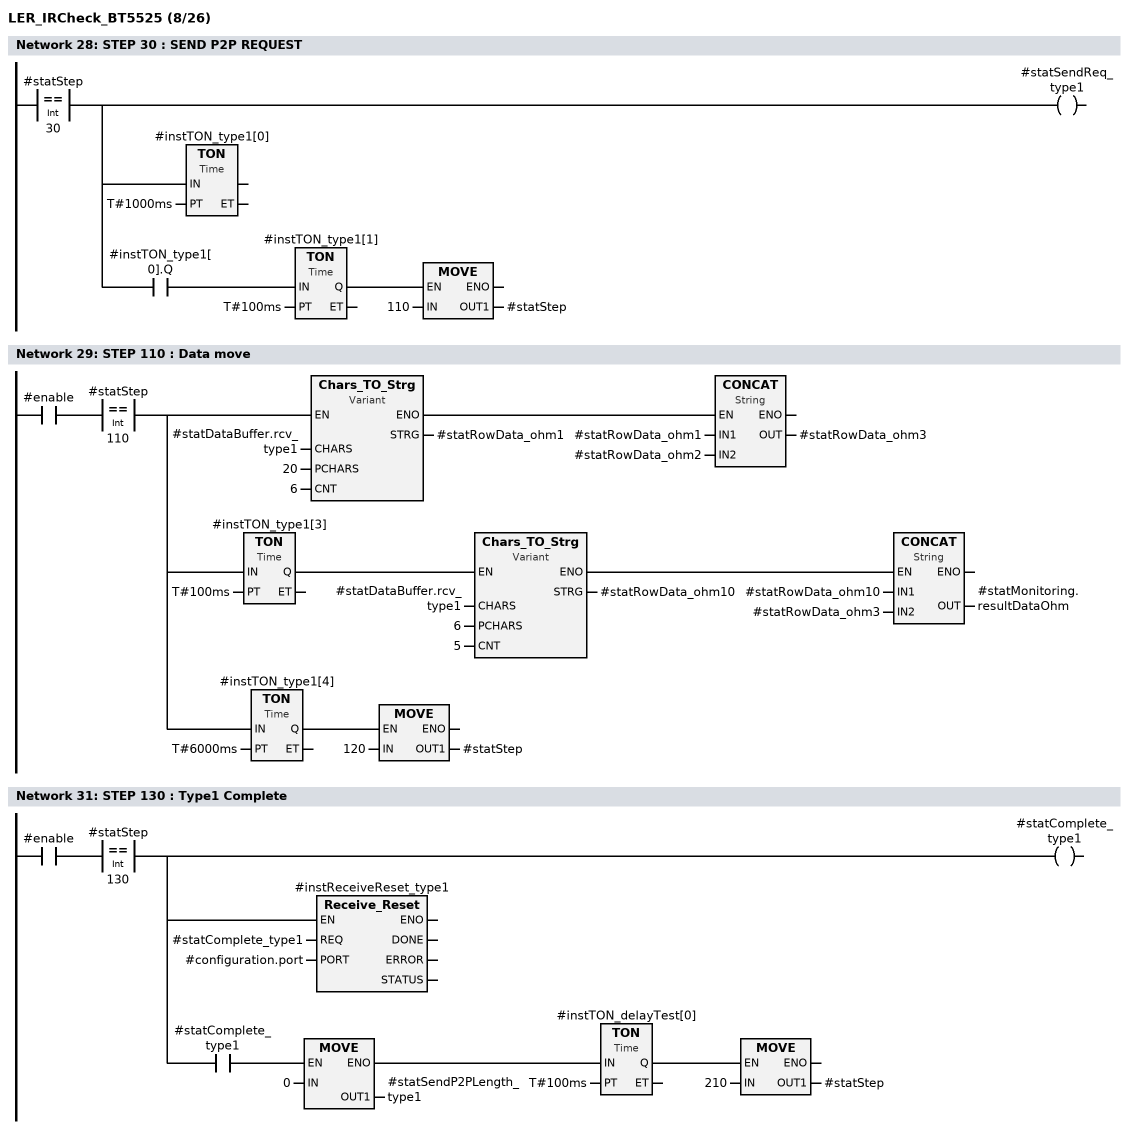
   RUNG wire#powerrail
      { S7_Templates := "SrcType := Int" } EQ_Contact(in1 := #statStep, in2 := 30)
      wire#w1
      Coil( #statSendReq_type1 )
   END_RUNG
   RUNG wire#w1
      { S7_Templates := "time_type := Time" } #instTON_type1[0].TON(pt := T#1000ms, et =>)
   END_RUNG
   RUNG wire#w1
      Contact( #instTON_type1[0].Q )
      { S7_Templates := "time_type := Time" } #instTON_type1[1].TON(pt := T#100ms, et =>)
      Move(in := 110, out1 => #statStep)
   END_RUNG
   // the same network as SCL:
   #statSendReq_type1 := #statStep = 30;
   #instTON_type1[0].TON(IN := #statSendReq_type1, PT := T#1000ms);
   #instTON_type1[1].TON(IN := #statSendReq_type1 AND #instTON_type1[0].Q, PT := T#100ms);
   IF #instTON_type1[1].Q THEN #statStep := 110; END_IF;
END_REGION

REGION Network 29: STEP 110 : Data move
   RUNG wire#powerrail
      Contact( #enable )
      { S7_Templates := "SrcType := Int" } EQ_Contact(in1 := #statStep, in2 := 110)
      wire#w1
      { S7_Templates := "[ptr_type := Variant, str_type := String]" } Chars_TO_Strg(Chars := #statDataBuffer.rcv_type1, pChars := 20, Cnt := 6, Strg => #statRowData_ohm1)
      { S7_Templates := "[card := 2, str_type := String]" } CONCAT(IN1 := #statRowData_ohm1, IN2 := #statRowData_ohm2, OUT => #statRowData_ohm3)
   END_RUNG
   RUNG wire#w1
      { S7_Templates := "time_type := Time" } #instTON_type1[3].TON(pt := T#100ms, et =>)
      { S7_Templates := "[ptr_type := Variant, str_type := String]" } Chars_TO_Strg(Chars := #statDataBuffer.rcv_type1, pChars := 6, Cnt := 5, Strg => #statRowData_ohm10)
      { S7_Templates := "[card := 2, str_type := String]" } CONCAT(IN1 := #statRowData_ohm10, IN2 := #statRowData_ohm3, OUT => #statMonitoring.resultDataOhm)
   END_RUNG
   RUNG wire#w1
      { S7_Templates := "time_type := Time" } #instTON_type1[4].TON(pt := T#6000ms, et =>)
      Move(in := 120, out1 => #statStep)
   END_RUNG
   // the same network as SCL:
   #_w1 := #enable AND (#statStep = 110);
   Chars_TO_Strg(EN := #_w1,
                 Chars := #statDataBuffer.rcv_type1,
                 pChars := 20,
                 Cnt := 6,
                 Strg => #statRowData_ohm1,
                 ENO => #_w2);
   IF #_w2 THEN CONCAT(IN1 := #statRowData_ohm1, IN2 := #statRowData_ohm2, OUT => #statRowData_ohm3); END_IF;
   #instTON_type1[3].TON(IN := #_w1, PT := T#100ms);
   Chars_TO_Strg(EN := #instTON_type1[3].Q,
                 Chars := #statDataBuffer.rcv_type1,
                 pChars := 6,
                 Cnt := 5,
                 Strg => #statRowData_ohm10,
                 ENO => #_w3);
   IF #_w3 THEN
       CONCAT(IN1 := #statRowData_ohm10, IN2 := #statRowData_ohm3, OUT => #statMonitoring.resultDataOhm);
   END_IF;
   #instTON_type1[4].TON(IN := #_w1, PT := T#6000ms);
   IF #instTON_type1[4].Q THEN #statStep := 120; END_IF;
END_REGION

REGION Network 30 (SCL): STEP 120 : Result check
   IF #enable THEN
       IF #statStep = 120 THEN
           // Error 기기 이상
           IF #statRowData_ohm1 = 'ERROR' THEN
               #statMonitoring.result := 8; // ERROR
           END_IF;

           // H.ERR 오버 히트 에러
           IF #statRowData_ohm1 = 'H.ERR' THEN
               #statMonitoring.result := 4; // ERROR
           END_IF;

           // O.F. 레인지 오버
           IF #statRowData_ohm1 = 'O.F.' THEN
               #statMonitoring.result := 5; // ERROR
           END_IF;

           // U.F. 레인지 언더
           IF #statRowData_ohm1 = 'ULFAIL' THEN
               #statMonitoring.result := 6; // ERROR
           END_IF;

           // C.ERR 컨택트 체크
           IF #statRowData_ohm1 = 'C.ERR' THEN
               #statMonitoring.result := 7; // ERROR
           END_IF;

           // INVAL 미측정
           IF #statRowData_ohm1 = 'INVAL' THEN
               #statMonitoring.result := 9; // ERROR
           END_IF;

           // NOCOMP 미판정 
           IF #statRowData_ohm10 = 'NOCOMP' THEN
               //#statRowData_ohm1 := '-';
               #statMonitoring.result := 10;
           END_IF;

           // UFAIL 상한치 초과 값
           IF #statRowData_ohm10 = 'UFAIL' THEN
               #statMonitoring.result := 2;
           END_IF;

           //LFAIL 하한치 미만 값
           IF #statRowData_ohm10 = 'LFAIL' THEN
               #statMonitoring.result := 3;
           END_IF;

           //PASS 기준 범위 내
           IF #statRowData_ohm10 = 'PASS' THEN
               #statMonitoring.result := 1;
           END_IF;

           #statStep := 130;
       END_IF;
   END_IF;
END_REGION

REGION Network 31: STEP 130 : Type1 Complete
   RUNG wire#powerrail
      Contact( #enable )
      { S7_Templates := "SrcType := Int" } EQ_Contact(in1 := #statStep, in2 := 130)
      wire#w1
      Coil( #statComplete_type1 )
   END_RUNG
   RUNG wire#w1
      #instReceiveReset_type1.Receive_Reset(REQ := #statComplete_type1, PORT := #configuration.port, DONE =>, ERROR =>, STATUS =>)
   END_RUNG
   RUNG wire#w1
      Contact( #statComplete_type1 )
      Move(in := 0, out1 => #statSendP2PLength_type1)
      { S7_Templates := "time_type := Time" } #instTON_delayTest[0].TON(pt := T#100ms, et =>)
      Move(in := 210, out1 => #statStep)
   END_RUNG
   // the same network as SCL:
   #statComplete_type1 := #enable AND (#statStep = 130);
   IF #statComplete_type1 THEN
       #instReceiveReset_type1(REQ := #statComplete_type1, PORT := #configuration.port);   // Receive_Reset
   END_IF;
   #_w1 := #statComplete_type1 AND #statComplete_type1;
   IF #_w1 THEN #statSendP2PLength_type1 := 0; END_IF;
   #instTON_delayTest[0].TON(IN := #_w1, PT := T#100ms);
   IF #instTON_delayTest[0].Q THEN #statStep := 210; END_IF;
END_REGION

REGION Network 32: ========================================== Sequence step 210 ~
END_REGION

REGION Network 33: STEP 210 : Contact check start
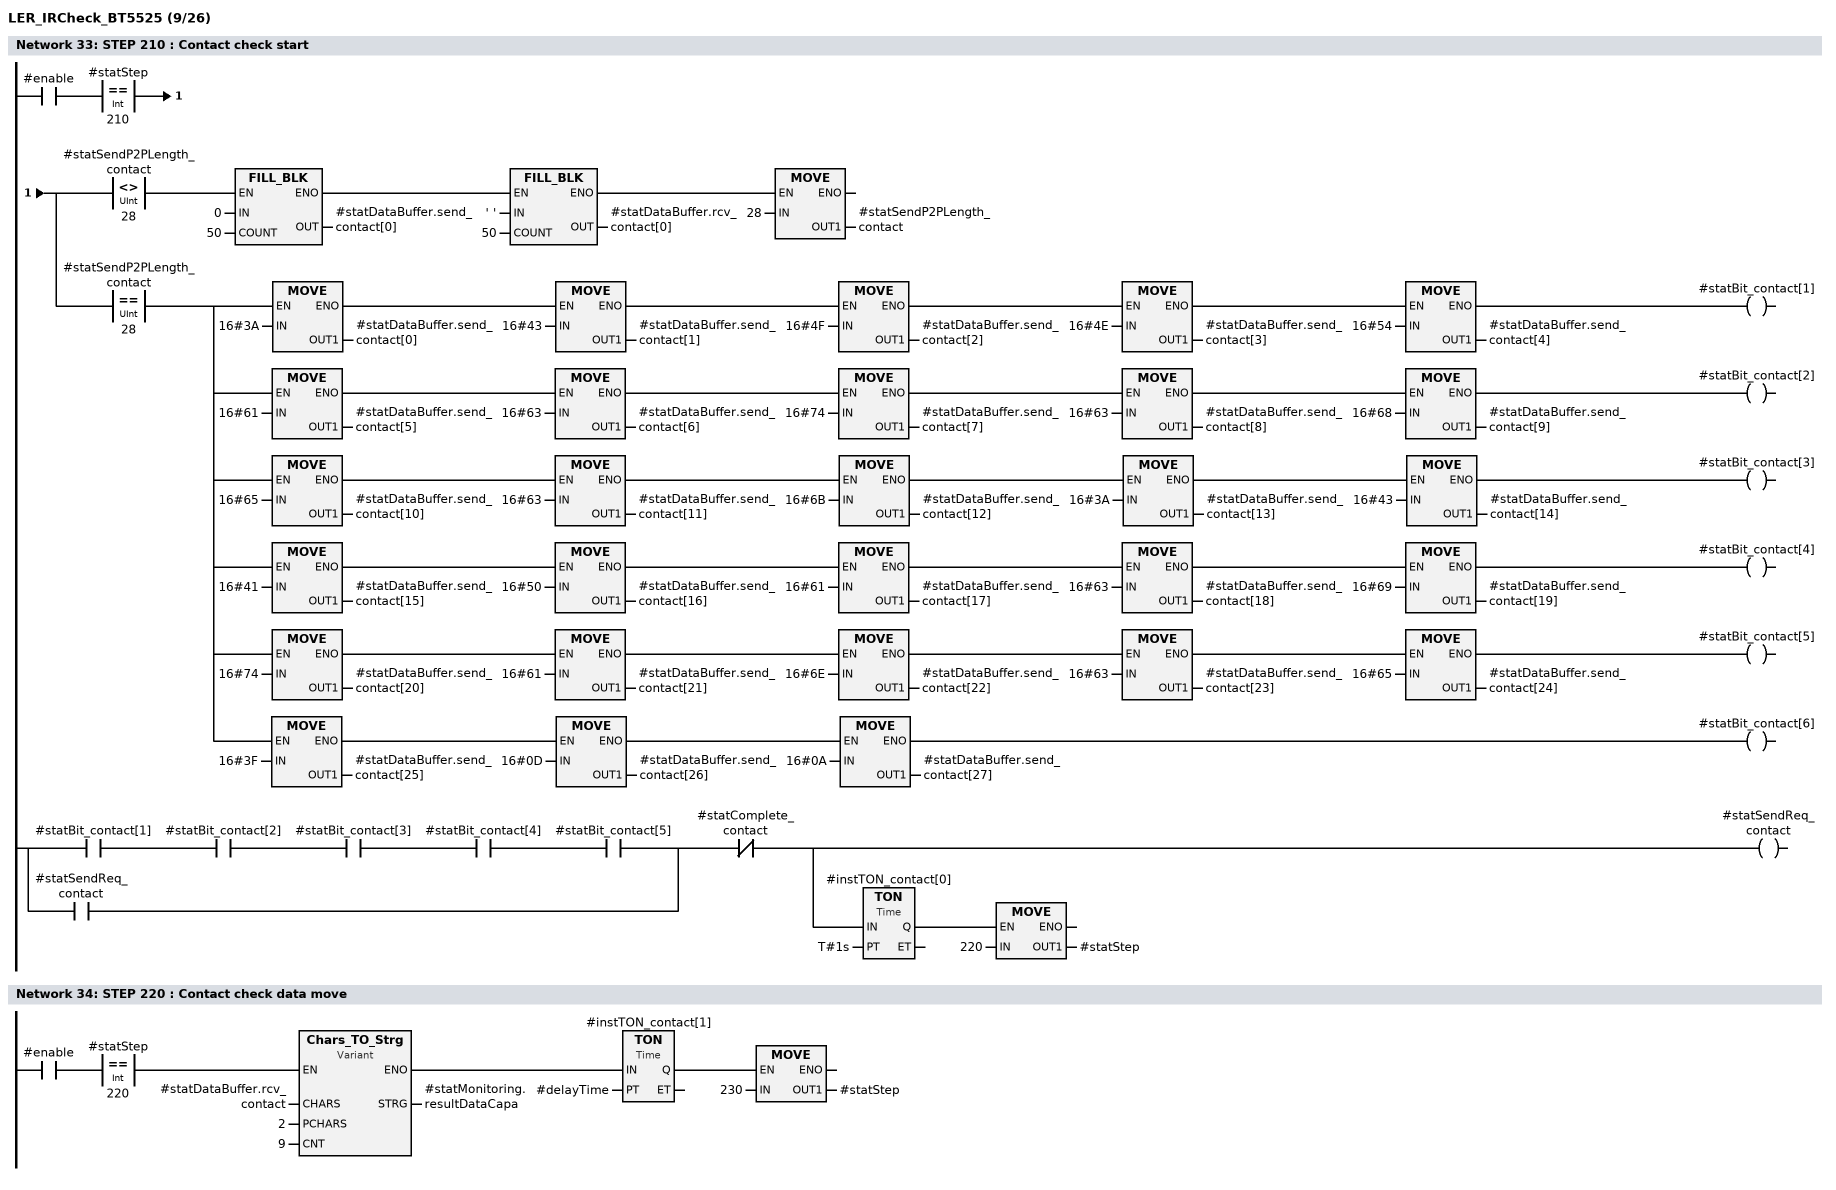
   RUNG wire#powerrail
      Contact( #enable )
      { S7_Templates := "SrcType := Int" } EQ_Contact(in1 := #statStep, in2 := 210)
      wire#w1
      { S7_Templates := "SrcType := UInt" } NE_Contact(in1 := #statSendP2PLength_contact, in2 := 28)
      FillBlockI(in := 0, count := 50, out => #statDataBuffer.send_contact[0])
      FillBlockI(in := ' ', count := 50, out => #statDataBuffer.rcv_contact[0])
      Move(in := 28, out1 => #statSendP2PLength_contact)
   END_RUNG
   RUNG wire#w1
      { S7_Templates := "SrcType := UInt" } EQ_Contact(in1 := #statSendP2PLength_contact, in2 := 28)
      wire#w2
      Move(in := 16#3A, out1 => #statDataBuffer.send_contact[0])
      Move(in := 16#43, out1 => #statDataBuffer.send_contact[1])
      Move(in := 16#4F, out1 => #statDataBuffer.send_contact[2])
      Move(in := 16#4E, out1 => #statDataBuffer.send_contact[3])
      Move(in := 16#54, out1 => #statDataBuffer.send_contact[4])
      Coil( #statBit_contact[1] )
   END_RUNG
   RUNG wire#w2
      Move(in := 16#61, out1 => #statDataBuffer.send_contact[5])
      Move(in := 16#63, out1 => #statDataBuffer.send_contact[6])
      Move(in := 16#74, out1 => #statDataBuffer.send_contact[7])
      Move(in := 16#63, out1 => #statDataBuffer.send_contact[8])
      Move(in := 16#68, out1 => #statDataBuffer.send_contact[9])
      Coil( #statBit_contact[2] )
   END_RUNG
   RUNG wire#w2
      Move(in := 16#65, out1 => #statDataBuffer.send_contact[10])
      Move(in := 16#63, out1 => #statDataBuffer.send_contact[11])
      Move(in := 16#6B, out1 => #statDataBuffer.send_contact[12])
      Move(in := 16#3A, out1 => #statDataBuffer.send_contact[13])
      Move(in := 16#43, out1 => #statDataBuffer.send_contact[14])
      Coil( #statBit_contact[3] )
   END_RUNG
   RUNG wire#w2
      Move(in := 16#41, out1 => #statDataBuffer.send_contact[15])
      Move(in := 16#50, out1 => #statDataBuffer.send_contact[16])
      Move(in := 16#61, out1 => #statDataBuffer.send_contact[17])
      Move(in := 16#63, out1 => #statDataBuffer.send_contact[18])
      Move(in := 16#69, out1 => #statDataBuffer.send_contact[19])
      Coil( #statBit_contact[4] )
   END_RUNG
   RUNG wire#w2
      Move(in := 16#74, out1 => #statDataBuffer.send_contact[20])
      Move(in := 16#61, out1 => #statDataBuffer.send_contact[21])
      Move(in := 16#6E, out1 => #statDataBuffer.send_contact[22])
      Move(in := 16#63, out1 => #statDataBuffer.send_contact[23])
      Move(in := 16#65, out1 => #statDataBuffer.send_contact[24])
      Coil( #statBit_contact[5] )
   END_RUNG
   RUNG wire#w2
      Move(in := 16#3F, out1 => #statDataBuffer.send_contact[25])
      Move(in := 16#0D, out1 => #statDataBuffer.send_contact[26])
      Move(in := 16#0A, out1 => #statDataBuffer.send_contact[27])
      Coil( #statBit_contact[6] )
   END_RUNG
   RUNG wire#powerrail
      Contact( #statBit_contact[1] )
      Contact( #statBit_contact[2] )
      Contact( #statBit_contact[3] )
      Contact( #statBit_contact[4] )
      Contact( #statBit_contact[5] )
      wire#w3
      I_Contact( #statComplete_contact )
      wire#w4
      Coil( #statSendReq_contact )
   END_RUNG
   RUNG wire#powerrail
      Contact( #statSendReq_contact )
   END_RUNG wire#w3
   RUNG wire#w4
      { S7_Templates := "time_type := Time" } #instTON_contact[0].TON(pt := T#1s, et =>)
      Move(in := 220, out1 => #statStep)
   END_RUNG
   // the same network as SCL:
   #_w1 := #enable AND (#statStep = 210);
   IF #_w1 AND (#statSendP2PLength_contact <> 28) THEN
       FILL_BLK(IN := 0, COUNT := 50, OUT => #statDataBuffer.send_contact[0]);
       FILL_BLK(IN := ' ', COUNT := 50, OUT => #statDataBuffer.rcv_contact[0]);
       #statSendP2PLength_contact := 28;
   END_IF;
   #_w2 := #_w1 AND (#statSendP2PLength_contact = 28);
   IF #_w2 THEN
       #statDataBuffer.send_contact[0] := 16#3A;
       #statDataBuffer.send_contact[1] := 16#43;
       #statDataBuffer.send_contact[2] := 16#4F;
       #statDataBuffer.send_contact[3] := 16#4E;
       #statDataBuffer.send_contact[4] := 16#54;
   END_IF;
   #statBit_contact[1] := #_w2;
   IF #_w2 THEN
       #statDataBuffer.send_contact[5] := 16#61;
       #statDataBuffer.send_contact[6] := 16#63;
       #statDataBuffer.send_contact[7] := 16#74;
       #statDataBuffer.send_contact[8] := 16#63;
       #statDataBuffer.send_contact[9] := 16#68;
   END_IF;
   #statBit_contact[2] := #_w2;
   IF #_w2 THEN
       #statDataBuffer.send_contact[10] := 16#65;
       #statDataBuffer.send_contact[11] := 16#63;
       #statDataBuffer.send_contact[12] := 16#6B;
       #statDataBuffer.send_contact[13] := 16#3A;
       #statDataBuffer.send_contact[14] := 16#43;
   END_IF;
   #statBit_contact[3] := #_w2;
   IF #_w2 THEN
       #statDataBuffer.send_contact[15] := 16#41;
       #statDataBuffer.send_contact[16] := 16#50;
       #statDataBuffer.send_contact[17] := 16#61;
       #statDataBuffer.send_contact[18] := 16#63;
       #statDataBuffer.send_contact[19] := 16#69;
   END_IF;
   #statBit_contact[4] := #_w2;
   IF #_w2 THEN
       #statDataBuffer.send_contact[20] := 16#74;
       #statDataBuffer.send_contact[21] := 16#61;
       #statDataBuffer.send_contact[22] := 16#6E;
       #statDataBuffer.send_contact[23] := 16#63;
       #statDataBuffer.send_contact[24] := 16#65;
   END_IF;
   #statBit_contact[5] := #_w2;
   IF #_w2 THEN
       #statDataBuffer.send_contact[25] := 16#3F;
       #statDataBuffer.send_contact[26] := 16#0D;
       #statDataBuffer.send_contact[27] := 16#0A;
   END_IF;
   #statBit_contact[6] := #_w2;
   #statSendReq_contact := ((#statBit_contact[1] AND #statBit_contact[2] AND #statBit_contact[3] AND #statBit_contact[4] AND #statBit_contact[5]) OR #statSendReq_contact) AND NOT #statComplete_contact;
   #instTON_contact[0].TON(IN := #statSendReq_contact, PT := T#1s);
   IF #instTON_contact[0].Q THEN #statStep := 220; END_IF;
END_REGION

REGION Network 34: STEP 220 : Contact check data move
   RUNG wire#powerrail
      Contact( #enable )
      { S7_Templates := "SrcType := Int" } EQ_Contact(in1 := #statStep, in2 := 220)
      { S7_Templates := "[ptr_type := Variant, str_type := String]" } Chars_TO_Strg(Chars := #statDataBuffer.rcv_contact, pChars := 2, Cnt := 9, Strg => #statMonitoring.resultDataCapa)
      { S7_Templates := "time_type := Time" } #instTON_contact[1].TON(pt := #delayTime, et =>)
      Move(in := 230, out1 => #statStep)
   END_RUNG
   // the same network as SCL:
   #_w1 := #enable AND (#statStep = 220);
   Chars_TO_Strg(EN := #_w1,
                 Chars := #statDataBuffer.rcv_contact,
                 pChars := 2,
                 Cnt := 9,
                 Strg => #statMonitoring.resultDataCapa,
                 ENO => #_w2);
   #instTON_contact[1].TON(IN := #_w2, PT := #delayTime);
   IF #instTON_contact[1].Q THEN #statStep := 230; END_IF;
END_REGION

REGION Network 35: STEP 230 : Contact check complete
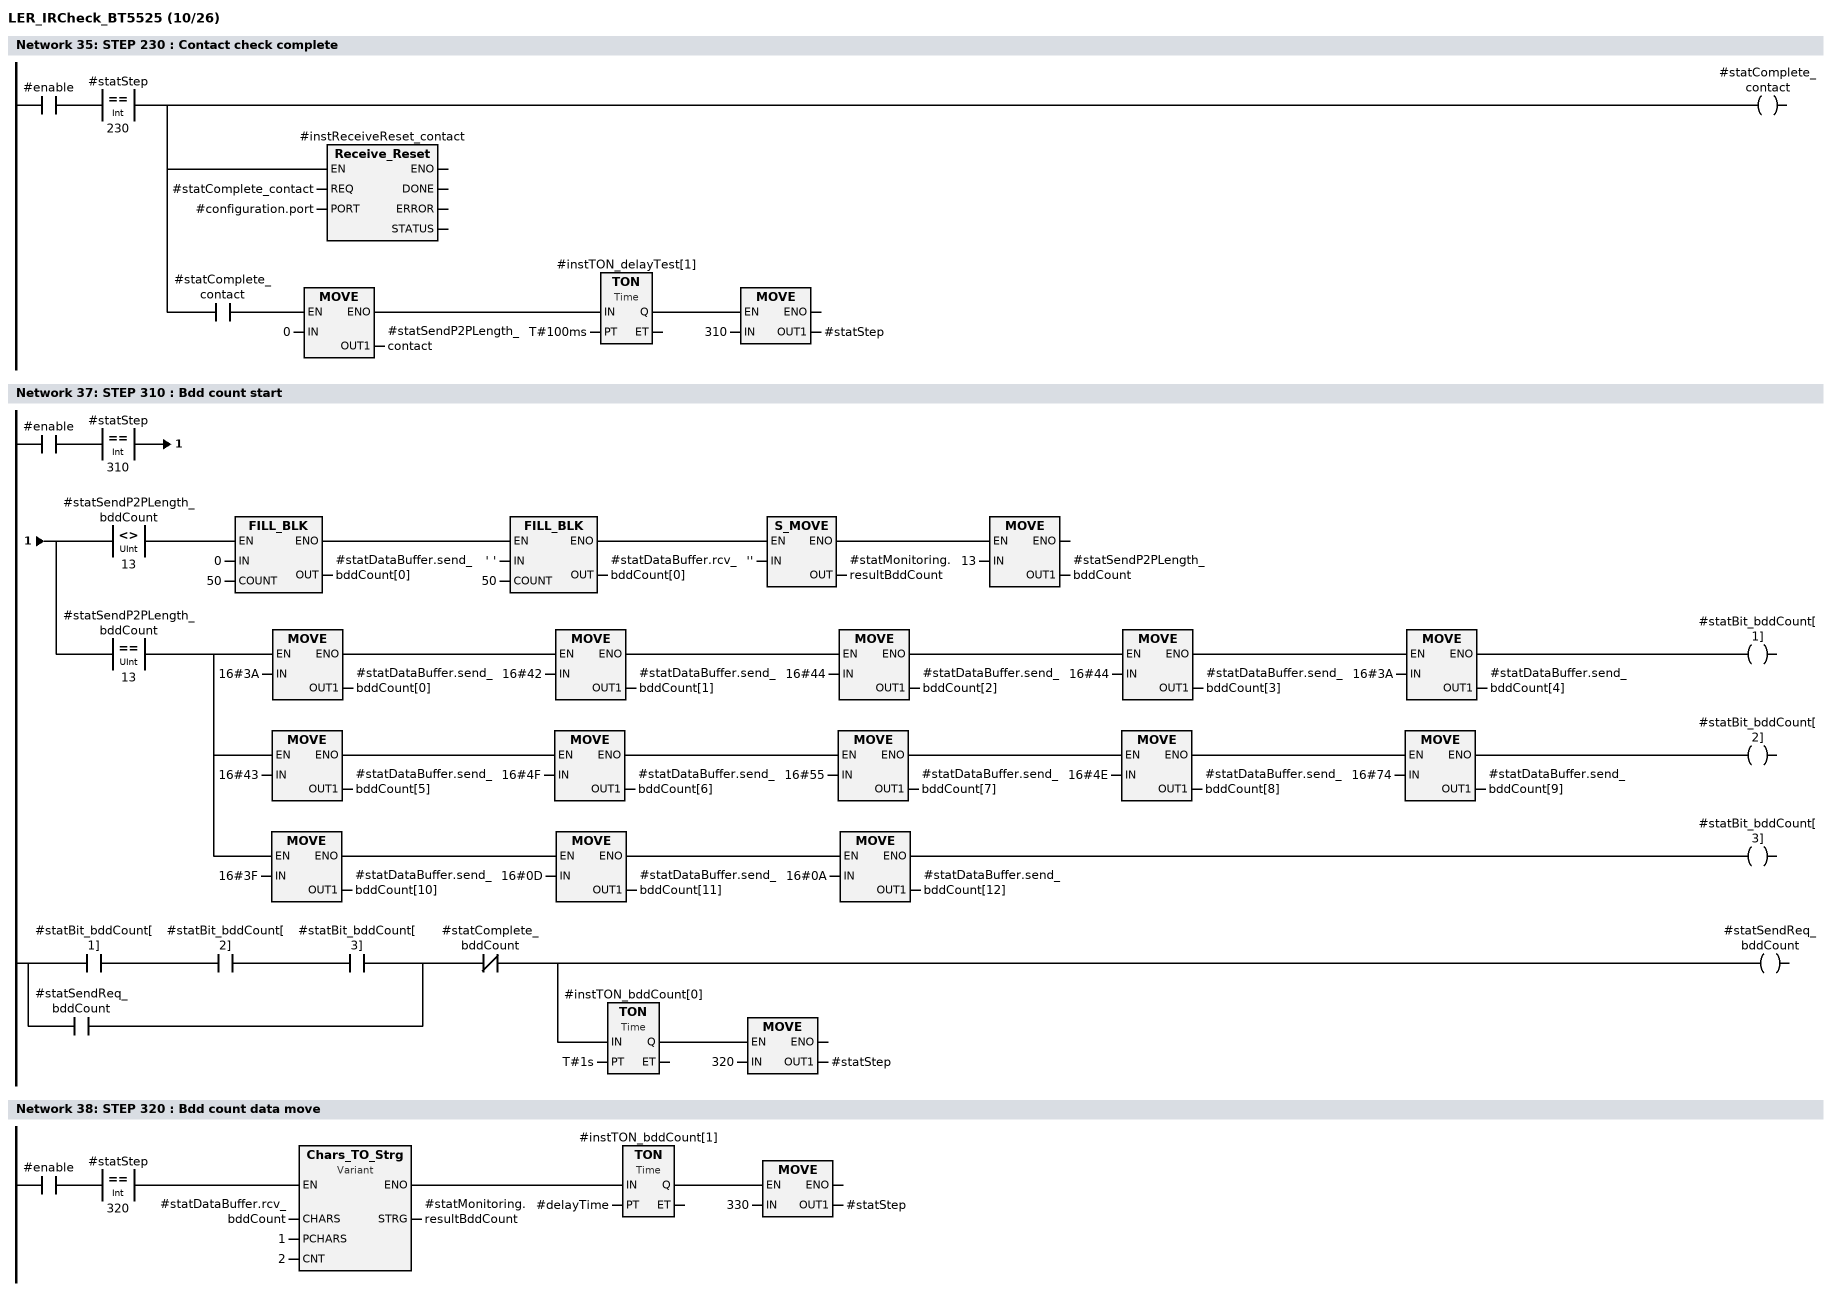
   RUNG wire#powerrail
      Contact( #enable )
      { S7_Templates := "SrcType := Int" } EQ_Contact(in1 := #statStep, in2 := 230)
      wire#w1
      Coil( #statComplete_contact )
   END_RUNG
   RUNG wire#w1
      #instReceiveReset_contact.Receive_Reset(REQ := #statComplete_contact, PORT := #configuration.port, DONE =>, ERROR =>, STATUS =>)
   END_RUNG
   RUNG wire#w1
      Contact( #statComplete_contact )
      Move(in := 0, out1 => #statSendP2PLength_contact)
      { S7_Templates := "time_type := Time" } #instTON_delayTest[1].TON(pt := T#100ms, et =>)
      Move(in := 310, out1 => #statStep)
   END_RUNG
   // the same network as SCL:
   #statComplete_contact := #enable AND (#statStep = 230);
   IF #statComplete_contact THEN
       #instReceiveReset_contact(REQ := #statComplete_contact, PORT := #configuration.port);   // Receive_Reset
   END_IF;
   #_w1 := #statComplete_contact AND #statComplete_contact;
   IF #_w1 THEN #statSendP2PLength_contact := 0; END_IF;
   #instTON_delayTest[1].TON(IN := #_w1, PT := T#100ms);
   IF #instTON_delayTest[1].Q THEN #statStep := 310; END_IF;
END_REGION

REGION Network 36: ========================================== Sequence step 310 ~
END_REGION

REGION Network 37: STEP 310 : Bdd count start
   RUNG wire#powerrail
      Contact( #enable )
      { S7_Templates := "SrcType := Int" } EQ_Contact(in1 := #statStep, in2 := 310)
      wire#w1
      { S7_Templates := "SrcType := UInt" } NE_Contact(in1 := #statSendP2PLength_bddCount, in2 := 13)
      FillBlockI(in := 0, count := 50, out => #statDataBuffer.send_bddCount[0])
      FillBlockI(in := ' ', count := 50, out => #statDataBuffer.rcv_bddCount[0])
      S_Move(in := '', out => #statMonitoring.resultBddCount)
      Move(in := 13, out1 => #statSendP2PLength_bddCount)
   END_RUNG
   RUNG wire#w1
      { S7_Templates := "SrcType := UInt" } EQ_Contact(in1 := #statSendP2PLength_bddCount, in2 := 13)
      wire#w2
      Move(in := 16#3A, out1 => #statDataBuffer.send_bddCount[0])
      Move(in := 16#42, out1 => #statDataBuffer.send_bddCount[1])
      Move(in := 16#44, out1 => #statDataBuffer.send_bddCount[2])
      Move(in := 16#44, out1 => #statDataBuffer.send_bddCount[3])
      Move(in := 16#3A, out1 => #statDataBuffer.send_bddCount[4])
      Coil( #statBit_bddCount[1] )
   END_RUNG
   RUNG wire#w2
      Move(in := 16#43, out1 => #statDataBuffer.send_bddCount[5])
      Move(in := 16#4F, out1 => #statDataBuffer.send_bddCount[6])
      Move(in := 16#55, out1 => #statDataBuffer.send_bddCount[7])
      Move(in := 16#4E, out1 => #statDataBuffer.send_bddCount[8])
      Move(in := 16#74, out1 => #statDataBuffer.send_bddCount[9])
      Coil( #statBit_bddCount[2] )
   END_RUNG
   RUNG wire#w2
      Move(in := 16#3F, out1 => #statDataBuffer.send_bddCount[10])
      Move(in := 16#0D, out1 => #statDataBuffer.send_bddCount[11])
      Move(in := 16#0A, out1 => #statDataBuffer.send_bddCount[12])
      Coil( #statBit_bddCount[3] )
   END_RUNG
   RUNG wire#powerrail
      Contact( #statBit_bddCount[1] )
      Contact( #statBit_bddCount[2] )
      Contact( #statBit_bddCount[3] )
      wire#w3
      I_Contact( #statComplete_bddCount )
      wire#w4
      Coil( #statSendReq_bddCount )
   END_RUNG
   RUNG wire#powerrail
      Contact( #statSendReq_bddCount )
   END_RUNG wire#w3
   RUNG wire#w4
      { S7_Templates := "time_type := Time" } #instTON_bddCount[0].TON(pt := T#1s, et =>)
      Move(in := 320, out1 => #statStep)
   END_RUNG
   // the same network as SCL:
   #_w1 := #enable AND (#statStep = 310);
   IF #_w1 AND (#statSendP2PLength_bddCount <> 13) THEN
       FILL_BLK(IN := 0, COUNT := 50, OUT => #statDataBuffer.send_bddCount[0]);
       FILL_BLK(IN := ' ', COUNT := 50, OUT => #statDataBuffer.rcv_bddCount[0]);
       #statMonitoring.resultBddCount := '';
       #statSendP2PLength_bddCount := 13;
   END_IF;
   #_w2 := #_w1 AND (#statSendP2PLength_bddCount = 13);
   IF #_w2 THEN
       #statDataBuffer.send_bddCount[0] := 16#3A;
       #statDataBuffer.send_bddCount[1] := 16#42;
       #statDataBuffer.send_bddCount[2] := 16#44;
       #statDataBuffer.send_bddCount[3] := 16#44;
       #statDataBuffer.send_bddCount[4] := 16#3A;
   END_IF;
   #statBit_bddCount[1] := #_w2;
   IF #_w2 THEN
       #statDataBuffer.send_bddCount[5] := 16#43;
       #statDataBuffer.send_bddCount[6] := 16#4F;
       #statDataBuffer.send_bddCount[7] := 16#55;
       #statDataBuffer.send_bddCount[8] := 16#4E;
       #statDataBuffer.send_bddCount[9] := 16#74;
   END_IF;
   #statBit_bddCount[2] := #_w2;
   IF #_w2 THEN
       #statDataBuffer.send_bddCount[10] := 16#3F;
       #statDataBuffer.send_bddCount[11] := 16#0D;
       #statDataBuffer.send_bddCount[12] := 16#0A;
   END_IF;
   #statBit_bddCount[3] := #_w2;
   #statSendReq_bddCount := ((#statBit_bddCount[1] AND #statBit_bddCount[2] AND #statBit_bddCount[3]) OR #statSendReq_bddCount) AND NOT #statComplete_bddCount;
   #instTON_bddCount[0].TON(IN := #statSendReq_bddCount, PT := T#1s);
   IF #instTON_bddCount[0].Q THEN #statStep := 320; END_IF;
END_REGION

REGION Network 38: STEP 320 : Bdd count data move
   RUNG wire#powerrail
      Contact( #enable )
      { S7_Templates := "SrcType := Int" } EQ_Contact(in1 := #statStep, in2 := 320)
      { S7_Templates := "[ptr_type := Variant, str_type := String]" } Chars_TO_Strg(Chars := #statDataBuffer.rcv_bddCount, pChars := 1, Cnt := 2, Strg => #statMonitoring.resultBddCount)
      { S7_Templates := "time_type := Time" } #instTON_bddCount[1].TON(pt := #delayTime, et =>)
      Move(in := 330, out1 => #statStep)
   END_RUNG
   // the same network as SCL:
   #_w1 := #enable AND (#statStep = 320);
   Chars_TO_Strg(EN := #_w1,
                 Chars := #statDataBuffer.rcv_bddCount,
                 pChars := 1,
                 Cnt := 2,
                 Strg => #statMonitoring.resultBddCount,
                 ENO => #_w2);
   #instTON_bddCount[1].TON(IN := #_w2, PT := #delayTime);
   IF #instTON_bddCount[1].Q THEN #statStep := 330; END_IF;
END_REGION

REGION Network 39: STEP 330 : Bdd count complete
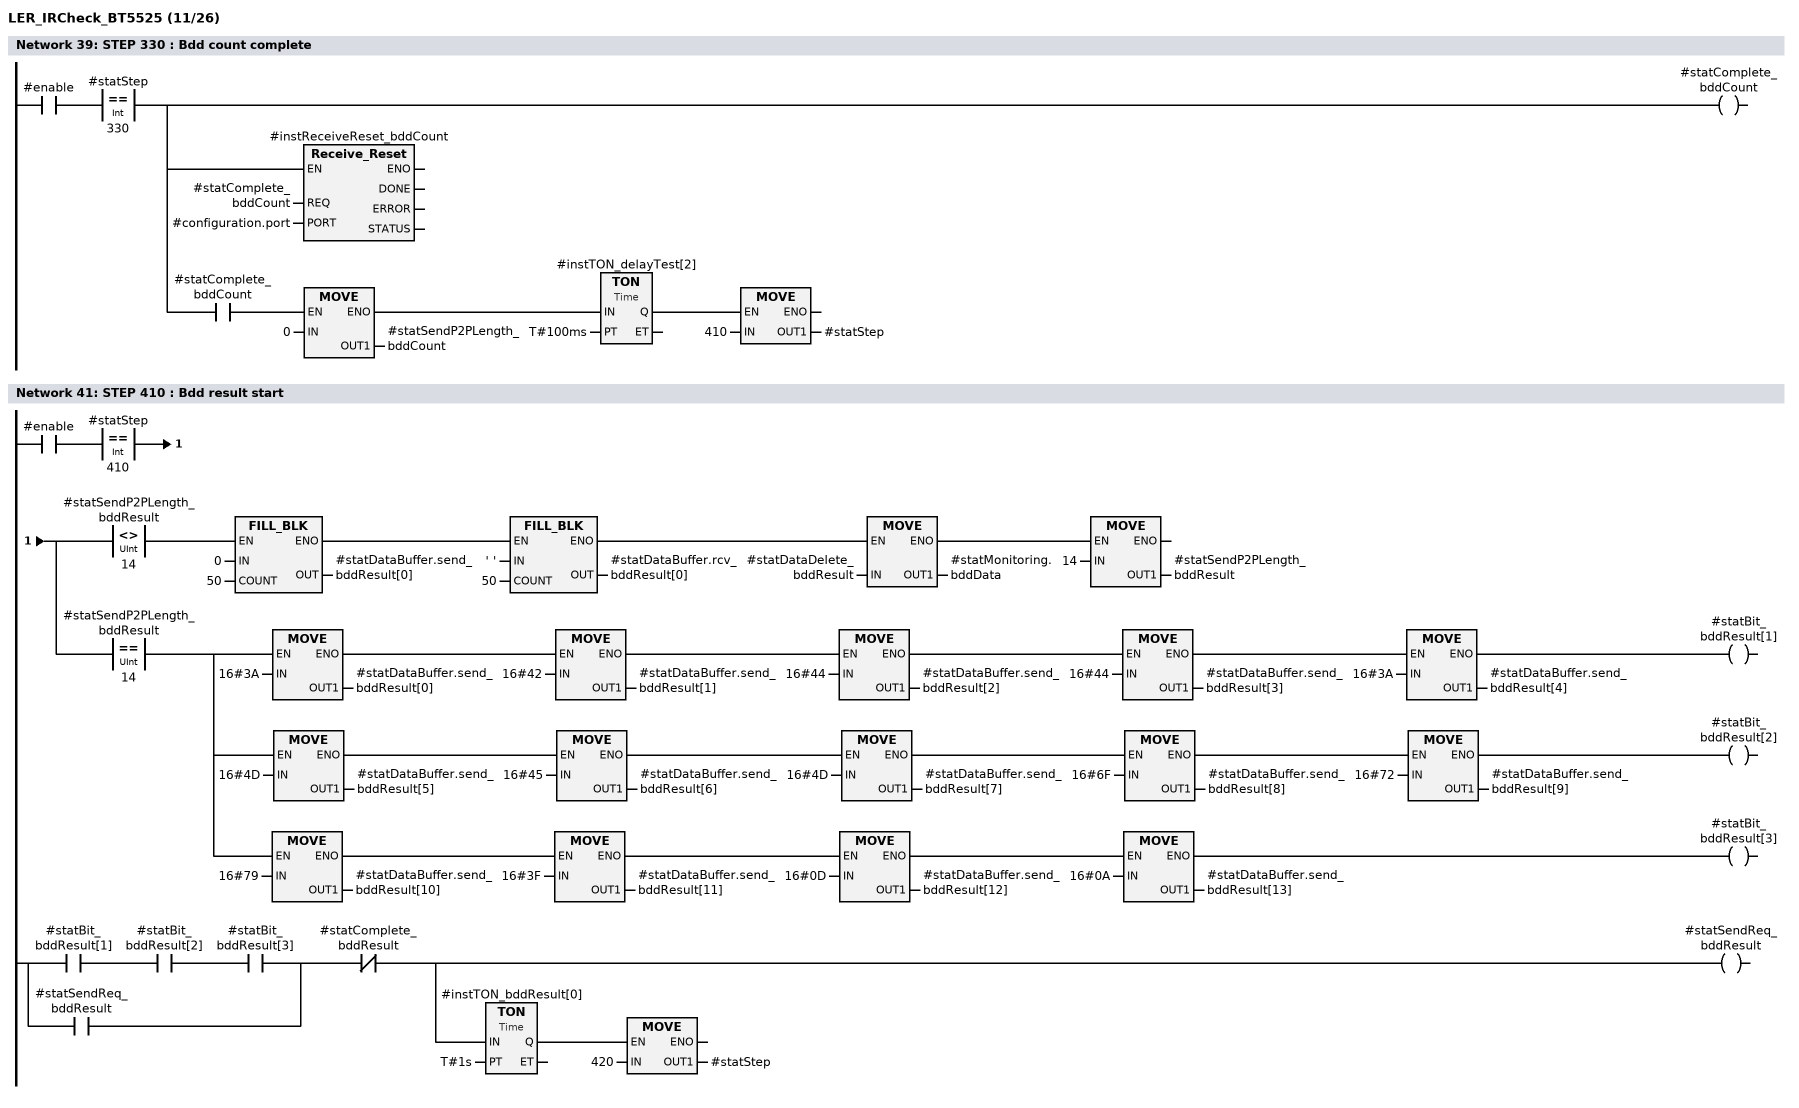
   RUNG wire#powerrail
      Contact( #enable )
      { S7_Templates := "SrcType := Int" } EQ_Contact(in1 := #statStep, in2 := 330)
      wire#w1
      Coil( #statComplete_bddCount )
   END_RUNG
   RUNG wire#w1
      #instReceiveReset_bddCount.Receive_Reset(REQ := #statComplete_bddCount, PORT := #configuration.port, DONE =>, ERROR =>, STATUS =>)
   END_RUNG
   RUNG wire#w1
      Contact( #statComplete_bddCount )
      Move(in := 0, out1 => #statSendP2PLength_bddCount)
      { S7_Templates := "time_type := Time" } #instTON_delayTest[2].TON(pt := T#100ms, et =>)
      Move(in := 410, out1 => #statStep)
   END_RUNG
   // the same network as SCL:
   #statComplete_bddCount := #enable AND (#statStep = 330);
   IF #statComplete_bddCount THEN
       #instReceiveReset_bddCount(REQ := #statComplete_bddCount, PORT := #configuration.port);   // Receive_Reset
   END_IF;
   #_w1 := #statComplete_bddCount AND #statComplete_bddCount;
   IF #_w1 THEN #statSendP2PLength_bddCount := 0; END_IF;
   #instTON_delayTest[2].TON(IN := #_w1, PT := T#100ms);
   IF #instTON_delayTest[2].Q THEN #statStep := 410; END_IF;
END_REGION

REGION Network 40: ========================================== Sequence step 410 ~
END_REGION

REGION Network 41: STEP 410 : Bdd result start
   RUNG wire#powerrail
      Contact( #enable )
      { S7_Templates := "SrcType := Int" } EQ_Contact(in1 := #statStep, in2 := 410)
      wire#w1
      { S7_Templates := "SrcType := UInt" } NE_Contact(in1 := #statSendP2PLength_bddResult, in2 := 14)
      FillBlockI(in := 0, count := 50, out => #statDataBuffer.send_bddResult[0])
      FillBlockI(in := ' ', count := 50, out => #statDataBuffer.rcv_bddResult[0])
      Move(in := #statDataDelete_bddResult, out1 => #statMonitoring.bddData)
      Move(in := 14, out1 => #statSendP2PLength_bddResult)
   END_RUNG
   RUNG wire#w1
      { S7_Templates := "SrcType := UInt" } EQ_Contact(in1 := #statSendP2PLength_bddResult, in2 := 14)
      wire#w2
      Move(in := 16#3A, out1 => #statDataBuffer.send_bddResult[0])
      Move(in := 16#42, out1 => #statDataBuffer.send_bddResult[1])
      Move(in := 16#44, out1 => #statDataBuffer.send_bddResult[2])
      Move(in := 16#44, out1 => #statDataBuffer.send_bddResult[3])
      Move(in := 16#3A, out1 => #statDataBuffer.send_bddResult[4])
      Coil( #statBit_bddResult[1] )
   END_RUNG
   RUNG wire#w2
      Move(in := 16#4D, out1 => #statDataBuffer.send_bddResult[5])
      Move(in := 16#45, out1 => #statDataBuffer.send_bddResult[6])
      Move(in := 16#4D, out1 => #statDataBuffer.send_bddResult[7])
      Move(in := 16#6F, out1 => #statDataBuffer.send_bddResult[8])
      Move(in := 16#72, out1 => #statDataBuffer.send_bddResult[9])
      Coil( #statBit_bddResult[2] )
   END_RUNG
   RUNG wire#w2
      Move(in := 16#79, out1 => #statDataBuffer.send_bddResult[10])
      Move(in := 16#3F, out1 => #statDataBuffer.send_bddResult[11])
      Move(in := 16#0D, out1 => #statDataBuffer.send_bddResult[12])
      Move(in := 16#0A, out1 => #statDataBuffer.send_bddResult[13])
      Coil( #statBit_bddResult[3] )
   END_RUNG
   RUNG wire#powerrail
      Contact( #statBit_bddResult[1] )
      Contact( #statBit_bddResult[2] )
      Contact( #statBit_bddResult[3] )
      wire#w3
      I_Contact( #statComplete_bddResult )
      wire#w4
      Coil( #statSendReq_bddResult )
   END_RUNG
   RUNG wire#powerrail
      Contact( #statSendReq_bddResult )
   END_RUNG wire#w3
   RUNG wire#w4
      { S7_Templates := "time_type := Time" } #instTON_bddResult[0].TON(pt := T#1s, et =>)
      Move(in := 420, out1 => #statStep)
   END_RUNG
   // the same network as SCL:
   #_w1 := #enable AND (#statStep = 410);
   IF #_w1 AND (#statSendP2PLength_bddResult <> 14) THEN
       FILL_BLK(IN := 0, COUNT := 50, OUT => #statDataBuffer.send_bddResult[0]);
       FILL_BLK(IN := ' ', COUNT := 50, OUT => #statDataBuffer.rcv_bddResult[0]);
       #statMonitoring.bddData := #statDataDelete_bddResult;
       #statSendP2PLength_bddResult := 14;
   END_IF;
   #_w2 := #_w1 AND (#statSendP2PLength_bddResult = 14);
   IF #_w2 THEN
       #statDataBuffer.send_bddResult[0] := 16#3A;
       #statDataBuffer.send_bddResult[1] := 16#42;
       #statDataBuffer.send_bddResult[2] := 16#44;
       #statDataBuffer.send_bddResult[3] := 16#44;
       #statDataBuffer.send_bddResult[4] := 16#3A;
   END_IF;
   #statBit_bddResult[1] := #_w2;
   IF #_w2 THEN
       #statDataBuffer.send_bddResult[5] := 16#4D;
       #statDataBuffer.send_bddResult[6] := 16#45;
       #statDataBuffer.send_bddResult[7] := 16#4D;
       #statDataBuffer.send_bddResult[8] := 16#6F;
       #statDataBuffer.send_bddResult[9] := 16#72;
   END_IF;
   #statBit_bddResult[2] := #_w2;
   IF #_w2 THEN
       #statDataBuffer.send_bddResult[10] := 16#79;
       #statDataBuffer.send_bddResult[11] := 16#3F;
       #statDataBuffer.send_bddResult[12] := 16#0D;
       #statDataBuffer.send_bddResult[13] := 16#0A;
   END_IF;
   #statBit_bddResult[3] := #_w2;
   #statSendReq_bddResult := ((#statBit_bddResult[1] AND #statBit_bddResult[2] AND #statBit_bddResult[3]) OR #statSendReq_bddResult) AND NOT #statComplete_bddResult;
   #instTON_bddResult[0].TON(IN := #statSendReq_bddResult, PT := T#1s);
   IF #instTON_bddResult[0].Q THEN #statStep := 420; END_IF;
END_REGION

REGION Network 42 (SCL): STEP 420 : Bdd count data move
   IF #enable AND #statStep = 420 THEN
       //BDD Mode Of BDD Result Data
       Chars_TO_Strg(Chars := #statDataBuffer.rcv_bddResult,
                     pChars := 11,
                     Cnt := 3,
                     Strg => #statMonitoring.bddData.dataMode[0]);
       Chars_TO_Strg(Chars := #statDataBuffer.rcv_bddResult,
                     pChars := 35,
                     Cnt := 3,
                     Strg => #statMonitoring.bddData.dataMode[1]);
       Chars_TO_Strg(Chars := #statDataBuffer.rcv_bddResult,
                     pChars := 59,
                     Cnt := 3,
                     Strg => #statMonitoring.bddData.dataMode[2]);
       Chars_TO_Strg(Chars := #statDataBuffer.rcv_bddResult,
                     pChars := 83,
                     Cnt := 3,
                     Strg => #statMonitoring.bddData.dataMode[3]);
       Chars_TO_Strg(Chars := #statDataBuffer.rcv_bddResult,
                     pChars := 107,
                     Cnt := 3,
                     Strg => #statMonitoring.bddData.dataMode[4]);
       Chars_TO_Strg(Chars := #statDataBuffer.rcv_bddResult,
                     pChars := 131,
                     Cnt := 3,
                     Strg => #statMonitoring.bddData.dataMode[5]);
       Chars_TO_Strg(Chars := #statDataBuffer.rcv_bddResult,
                     pChars := 155,
                     Cnt := 3,
                     Strg => #statMonitoring.bddData.dataMode[6]);
       Chars_TO_Strg(Chars := #statDataBuffer.rcv_bddResult,
                     pChars := 179,
                     Cnt := 3,
                     Strg => #statMonitoring.bddData.dataMode[7]);
       Chars_TO_Strg(Chars := #statDataBuffer.rcv_bddResult,
                     pChars := 203,
                     Cnt := 3,
                     Strg => #statMonitoring.bddData.dataMode[8]);
       Chars_TO_Strg(Chars := #statDataBuffer.rcv_bddResult,
                     pChars := 227,
                     Cnt := 3,
                     Strg => #statMonitoring.bddData.dataMode[9]);

       Chars_TO_Strg(Chars := #statDataBuffer.rcv_bddResult,
                     pChars := 251,
                     Cnt := 3,
                     Strg => #statMonitoring.bddData.dataMode[10]);
       Chars_TO_Strg(Chars := #statDataBuffer.rcv_bddResult,
                     pChars := 275,
                     Cnt := 3,
                     Strg => #statMonitoring.bddData.dataMode[11]);
       Chars_TO_Strg(Chars := #statDataBuffer.rcv_bddResult,
                     pChars := 299,
                     Cnt := 3,
                     Strg => #statMonitoring.bddData.dataMode[12]);
       Chars_TO_Strg(Chars := #statDataBuffer.rcv_bddResult,
                     pChars := 323,
                     Cnt := 3,
                     Strg => #statMonitoring.bddData.dataMode[13]);
       Chars_TO_Strg(Chars := #statDataBuffer.rcv_bddResult,
                     pChars := 347,
                     Cnt := 3,
                     Strg => #statMonitoring.bddData.dataMode[14]);
       Chars_TO_Strg(Chars := #statDataBuffer.rcv_bddResult,
                     pChars := 371,
                     Cnt := 3,
                     Strg => #statMonitoring.bddData.dataMode[15]);
       Chars_TO_Strg(Chars := #statDataBuffer.rcv_bddResult,
                     pChars := 395,
                     Cnt := 3,
                     Strg => #statMonitoring.bddData.dataMode[16]);
       Chars_TO_Strg(Chars := #statDataBuffer.rcv_bddResult,
                     pChars := 419,
                     Cnt := 3,
                     Strg => #statMonitoring.bddData.dataMode[17]);
       Chars_TO_Strg(Chars := #statDataBuffer.rcv_bddResult,
                     pChars := 443,
                     Cnt := 3,
                     Strg => #statMonitoring.bddData.dataMode[18]);
       Chars_TO_Strg(Chars := #statDataBuffer.rcv_bddResult,
                     pChars := 467,
                     Cnt := 3,
                     Strg => #statMonitoring.bddData.dataMode[19]);

       Chars_TO_Strg(Chars := #statDataBuffer.rcv_bddResult,
                     pChars := 491,
                     Cnt := 3,
                     Strg => #statMonitoring.bddData.dataMode[20]);
       Chars_TO_Strg(Chars := #statDataBuffer.rcv_bddResult,
                     pChars := 515,
                     Cnt := 3,
                     Strg => #statMonitoring.bddData.dataMode[21]);
       Chars_TO_Strg(Chars := #statDataBuffer.rcv_bddResult,
                     pChars := 539,
                     Cnt := 3,
                     Strg => #statMonitoring.bddData.dataMode[22]);
       Chars_TO_Strg(Chars := #statDataBuffer.rcv_bddResult,
                     pChars := 563,
                     Cnt := 3,
                     Strg => #statMonitoring.bddData.dataMode[23]);
       Chars_TO_Strg(Chars := #statDataBuffer.rcv_bddResult,
                     pChars := 587,
                     Cnt := 3,
                     Strg => #statMonitoring.bddData.dataMode[24]);
       Chars_TO_Strg(Chars := #statDataBuffer.rcv_bddResult,
                     pChars := 611,
                     Cnt := 3,
                     Strg => #statMonitoring.bddData.dataMode[25]);
       Chars_TO_Strg(Chars := #statDataBuffer.rcv_bddResult,
                     pChars := 635,
                     Cnt := 3,
                     Strg => #statMonitoring.bddData.dataMode[26]);
       Chars_TO_Strg(Chars := #statDataBuffer.rcv_bddResult,
                     pChars := 659,
                     Cnt := 3,
                     Strg => #statMonitoring.bddData.dataMode[27]);
       Chars_TO_Strg(Chars := #statDataBuffer.rcv_bddResult,
                     pChars := 683,
                     Cnt := 3,
                     Strg => #statMonitoring.bddData.dataMode[28]);
       Chars_TO_Strg(Chars := #statDataBuffer.rcv_bddResult,
                     pChars := 707,
                     Cnt := 3,
                     Strg => #statMonitoring.bddData.dataMode[29]);

       Chars_TO_Strg(Chars := #statDataBuffer.rcv_bddResult,
                     pChars := 731,
                     Cnt := 3,
                     Strg => #statMonitoring.bddData.dataMode[30]);
       Chars_TO_Strg(Chars := #statDataBuffer.rcv_bddResult,
                     pChars := 755,
                     Cnt := 3,
                     Strg => #statMonitoring.bddData.dataMode[31]);
       Chars_TO_Strg(Chars := #statDataBuffer.rcv_bddResult,
                     pChars := 779,
                     Cnt := 3,
                     Strg => #statMonitoring.bddData.dataMode[32]);
       Chars_TO_Strg(Chars := #statDataBuffer.rcv_bddResult,
                     pChars := 803,
                     Cnt := 3,
                     Strg => #statMonitoring.bddData.dataMode[33]);
       Chars_TO_Strg(Chars := #statDataBuffer.rcv_bddResult,
                     pChars := 827,
                     Cnt := 3,
                     Strg => #statMonitoring.bddData.dataMode[34]);
       Chars_TO_Strg(Chars := #statDataBuffer.rcv_bddResult,
                     pChars := 851,
                     Cnt := 3,
                     Strg => #statMonitoring.bddData.dataMode[35]);
       Chars_TO_Strg(Chars := #statDataBuffer.rcv_bddResult,
                     pChars := 875,
                     Cnt := 3,
                     Strg => #statMonitoring.bddData.dataMode[36]);
       Chars_TO_Strg(Chars := #statDataBuffer.rcv_bddResult,
                     pChars := 899,
                     Cnt := 3,
                     Strg => #statMonitoring.bddData.dataMode[37]);
       Chars_TO_Strg(Chars := #statDataBuffer.rcv_bddResult,
                     pChars := 923,
                     Cnt := 3,
                     Strg => #statMonitoring.bddData.dataMode[38]);
       Chars_TO_Strg(Chars := #statDataBuffer.rcv_bddResult,
                     pChars := 947,
                     Cnt := 3,
                     Strg => #statMonitoring.bddData.dataMode[39]);

       Chars_TO_Strg(Chars := #statDataBuffer.rcv_bddResult,
                     pChars := 971,
                     Cnt := 3,
                     Strg => #statMonitoring.bddData.dataMode[40]);
       Chars_TO_Strg(Chars := #statDataBuffer.rcv_bddResult,
                     pChars := 995,
                     Cnt := 3,
                     Strg => #statMonitoring.bddData.dataMode[41]);
       Chars_TO_Strg(Chars := #statDataBuffer.rcv_bddResult,
                     pChars := 1019,
                     Cnt := 3,
                     Strg => #statMonitoring.bddData.dataMode[42]);
       Chars_TO_Strg(Chars := #statDataBuffer.rcv_bddResult,
                     pChars := 1043,
                     Cnt := 3,
                     Strg => #statMonitoring.bddData.dataMode[43]);
       Chars_TO_Strg(Chars := #statDataBuffer.rcv_bddResult,
                     pChars := 1067,
                     Cnt := 3,
                     Strg => #statMonitoring.bddData.dataMode[44]);
       Chars_TO_Strg(Chars := #statDataBuffer.rcv_bddResult,
                     pChars := 1091,
                     Cnt := 3,
                     Strg => #statMonitoring.bddData.dataMode[45]);
       Chars_TO_Strg(Chars := #statDataBuffer.rcv_bddResult,
                     pChars := 1115,
                     Cnt := 3,
                     Strg => #statMonitoring.bddData.dataMode[46]);
       Chars_TO_Strg(Chars := #statDataBuffer.rcv_bddResult,
                     pChars := 1139,
                     Cnt := 3,
                     Strg => #statMonitoring.bddData.dataMode[47]);
       Chars_TO_Strg(Chars := #statDataBuffer.rcv_bddResult,
                     pChars := 1163,
                     Cnt := 3,
                     Strg => #statMonitoring.bddData.dataMode[48]);
       Chars_TO_Strg(Chars := #statDataBuffer.rcv_bddResult,
                     pChars := 1187,
                     Cnt := 3,
                     Strg => #statMonitoring.bddData.dataMode[49]);

       Chars_TO_Strg(Chars := #statDataBuffer.rcv_bddResult,
                     pChars := 1211,
                     Cnt := 3,
                     Strg => #statMonitoring.bddData.dataMode[50]);
       Chars_TO_Strg(Chars := #statDataBuffer.rcv_bddResult,
                     pChars := 1235,
                     Cnt := 3,
                     Strg => #statMonitoring.bddData.dataMode[51]);
       Chars_TO_Strg(Chars := #statDataBuffer.rcv_bddResult,
                     pChars := 1259,
                     Cnt := 3,
                     Strg => #statMonitoring.bddData.dataMode[52]);
       Chars_TO_Strg(Chars := #statDataBuffer.rcv_bddResult,
                     pChars := 1283,
                     Cnt := 3,
                     Strg => #statMonitoring.bddData.dataMode[53]);
       Chars_TO_Strg(Chars := #statDataBuffer.rcv_bddResult,
                     pChars := 1307,
                     Cnt := 3,
                     Strg => #statMonitoring.bddData.dataMode[54]);
       Chars_TO_Strg(Chars := #statDataBuffer.rcv_bddResult,
                     pChars := 1331,
                     Cnt := 3,
                     Strg => #statMonitoring.bddData.dataMode[55]);
       Chars_TO_Strg(Chars := #statDataBuffer.rcv_bddResult,
                     pChars := 1355,
                     Cnt := 3,
                     Strg => #statMonitoring.bddData.dataMode[56]);
       Chars_TO_Strg(Chars := #statDataBuffer.rcv_bddResult,
                     pChars := 1379,
                     Cnt := 3,
                     Strg => #statMonitoring.bddData.dataMode[57]);
       Chars_TO_Strg(Chars := #statDataBuffer.rcv_bddResult,
                     pChars := 1403,
                     Cnt := 3,
                     Strg => #statMonitoring.bddData.dataMode[58]);
       Chars_TO_Strg(Chars := #statDataBuffer.rcv_bddResult,
                     pChars := 1427,
                     Cnt := 3,
                     Strg => #statMonitoring.bddData.dataMode[59]);

       Chars_TO_Strg(Chars := #statDataBuffer.rcv_bddResult,
                     pChars := 1451,
                     Cnt := 3,
                     Strg => #statMonitoring.bddData.dataMode[60]);
       Chars_TO_Strg(Chars := #statDataBuffer.rcv_bddResult,
                     pChars := 1475,
                     Cnt := 3,
                     Strg => #statMonitoring.bddData.dataMode[61]);
       Chars_TO_Strg(Chars := #statDataBuffer.rcv_bddResult,
                     pChars := 1499,
                     Cnt := 3,
                     Strg => #statMonitoring.bddData.dataMode[62]);
       Chars_TO_Strg(Chars := #statDataBuffer.rcv_bddResult,
                     pChars := 1523,
                     Cnt := 3,
                     Strg => #statMonitoring.bddData.dataMode[63]);
       Chars_TO_Strg(Chars := #statDataBuffer.rcv_bddResult,
                     pChars := 1547,
                     Cnt := 3,
                     Strg => #statMonitoring.bddData.dataMode[64]);
       Chars_TO_Strg(Chars := #statDataBuffer.rcv_bddResult,
                     pChars := 1571,
                     Cnt := 3,
                     Strg => #statMonitoring.bddData.dataMode[65]);
       Chars_TO_Strg(Chars := #statDataBuffer.rcv_bddResult,
                     pChars := 1595,
                     Cnt := 3,
                     Strg => #statMonitoring.bddData.dataMode[66]);
       Chars_TO_Strg(Chars := #statDataBuffer.rcv_bddResult,
                     pChars := 1619,
                     Cnt := 3,
                     Strg => #statMonitoring.bddData.dataMode[67]);
       Chars_TO_Strg(Chars := #statDataBuffer.rcv_bddResult,
                     pChars := 1643,
                     Cnt := 3,
                     Strg => #statMonitoring.bddData.dataMode[68]);
       Chars_TO_Strg(Chars := #statDataBuffer.rcv_bddResult,
                     pChars := 1667,
                     Cnt := 3,
                     Strg => #statMonitoring.bddData.dataMode[69]);

       Chars_TO_Strg(Chars := #statDataBuffer.rcv_bddResult,
                     pChars := 1691,
                     Cnt := 3,
                     Strg => #statMonitoring.bddData.dataMode[70]);
       Chars_TO_Strg(Chars := #statDataBuffer.rcv_bddResult,
                     pChars := 1715,
                     Cnt := 3,
                     Strg => #statMonitoring.bddData.dataMode[71]);
       Chars_TO_Strg(Chars := #statDataBuffer.rcv_bddResult,
                     pChars := 1739,
                     Cnt := 3,
                     Strg => #statMonitoring.bddData.dataMode[72]);
       Chars_TO_Strg(Chars := #statDataBuffer.rcv_bddResult,
                     pChars := 1763,
                     Cnt := 3,
                     Strg => #statMonitoring.bddData.dataMode[73]);
       Chars_TO_Strg(Chars := #statDataBuffer.rcv_bddResult,
                     pChars := 1787,
                     Cnt := 3,
                     Strg => #statMonitoring.bddData.dataMode[74]);
       Chars_TO_Strg(Chars := #statDataBuffer.rcv_bddResult,
                     pChars := 1811,
                     Cnt := 3,
                     Strg => #statMonitoring.bddData.dataMode[75]);
       Chars_TO_Strg(Chars := #statDataBuffer.rcv_bddResult,
                     pChars := 1835,
                     Cnt := 3,
                     Strg => #statMonitoring.bddData.dataMode[76]);
       Chars_TO_Strg(Chars := #statDataBuffer.rcv_bddResult,
                     pChars := 1859,
                     Cnt := 3,
                     Strg => #statMonitoring.bddData.dataMode[77]);
       Chars_TO_Strg(Chars := #statDataBuffer.rcv_bddResult,
                     pChars := 1883,
                     Cnt := 3,
                     Strg => #statMonitoring.bddData.dataMode[78]);
       Chars_TO_Strg(Chars := #statDataBuffer.rcv_bddResult,
                     pChars := 1907,
                     Cnt := 3,
                     Strg => #statMonitoring.bddData.dataMode[79]);

       Chars_TO_Strg(Chars := #statDataBuffer.rcv_bddResult,
                     pChars := 1931,
                     Cnt := 3,
                     Strg => #statMonitoring.bddData.dataMode[80]);
       Chars_TO_Strg(Chars := #statDataBuffer.rcv_bddResult,
                     pChars := 1955,
                     Cnt := 3,
                     Strg => #statMonitoring.bddData.dataMode[81]);
       Chars_TO_Strg(Chars := #statDataBuffer.rcv_bddResult,
                     pChars := 1979,
                     Cnt := 3,
                     Strg => #statMonitoring.bddData.dataMode[82]);
       Chars_TO_Strg(Chars := #statDataBuffer.rcv_bddResult,
                     pChars := 2003,
                     Cnt := 3,
                     Strg => #statMonitoring.bddData.dataMode[83]);
       Chars_TO_Strg(Chars := #statDataBuffer.rcv_bddResult,
                     pChars := 2027,
                     Cnt := 3,
                     Strg => #statMonitoring.bddData.dataMode[84]);
       Chars_TO_Strg(Chars := #statDataBuffer.rcv_bddResult,
                     pChars := 2051,
                     Cnt := 3,
                     Strg => #statMonitoring.bddData.dataMode[85]);
       Chars_TO_Strg(Chars := #statDataBuffer.rcv_bddResult,
                     pChars := 2075,
                     Cnt := 3,
                     Strg => #statMonitoring.bddData.dataMode[86]);
       Chars_TO_Strg(Chars := #statDataBuffer.rcv_bddResult,
                     pChars := 2099,
                     Cnt := 3,
                     Strg => #statMonitoring.bddData.dataMode[87]);
       Chars_TO_Strg(Chars := #statDataBuffer.rcv_bddResult,
                     pChars := 2123,
                     Cnt := 3,
                     Strg => #statMonitoring.bddData.dataMode[88]);
       Chars_TO_Strg(Chars := #statDataBuffer.rcv_bddResult,
                     pChars := 2147,
                     Cnt := 3,
                     Strg => #statMonitoring.bddData.dataMode[89]);

       Chars_TO_Strg(Chars := #statDataBuffer.rcv_bddResult,
                     pChars := 2171,
                     Cnt := 3,
                     Strg => #statMonitoring.bddData.dataMode[90]);
       Chars_TO_Strg(Chars := #statDataBuffer.rcv_bddResult,
                     pChars := 2195,
                     Cnt := 3,
                     Strg => #statMonitoring.bddData.dataMode[91]);
       Chars_TO_Strg(Chars := #statDataBuffer.rcv_bddResult,
                     pChars := 2219,
                     Cnt := 3,
                     Strg => #statMonitoring.bddData.dataMode[92]);
       Chars_TO_Strg(Chars := #statDataBuffer.rcv_bddResult,
                     pChars := 2243,
                     Cnt := 3,
                     Strg => #statMonitoring.bddData.dataMode[93]);
       Chars_TO_Strg(Chars := #statDataBuffer.rcv_bddResult,
                     pChars := 2267,
                     Cnt := 3,
                     Strg => #statMonitoring.bddData.dataMode[94]);
       Chars_TO_Strg(Chars := #statDataBuffer.rcv_bddResult,
                     pChars := 2291,
                     Cnt := 3,
                     Strg => #statMonitoring.bddData.dataMode[95]);
       Chars_TO_Strg(Chars := #statDataBuffer.rcv_bddResult,
                     pChars := 2315,
                     Cnt := 3,
                     Strg => #statMonitoring.bddData.dataMode[96]);
       Chars_TO_Strg(Chars := #statDataBuffer.rcv_bddResult,
                     pChars := 2339,
                     Cnt := 3,
                     Strg => #statMonitoring.bddData.dataMode[97]);
       Chars_TO_Strg(Chars := #statDataBuffer.rcv_bddResult,
                     pChars := 2363,
                     Cnt := 3,
                     Strg => #statMonitoring.bddData.dataMode[98]);
       Chars_TO_Strg(Chars := #statDataBuffer.rcv_bddResult,
                     pChars := 2387,
                     Cnt := 3,
                     Strg => #statMonitoring.bddData.dataMode[99]);

       //BDD Value Of BDD Result Data
       Chars_TO_Strg(Chars := #statDataBuffer.rcv_bddResult,
                     pChars := 15,
                     Cnt := 8,
                     Strg => #statMonitoring.bddData.dataValue[0]);
       Chars_TO_Strg(Chars := #statDataBuffer.rcv_bddResult,
                     pChars := 39,
                     Cnt := 8,
                     Strg => #statMonitoring.bddData.dataValue[1]);
       Chars_TO_Strg(Chars := #statDataBuffer.rcv_bddResult,
                     pChars := 63,
                     Cnt := 8,
                     Strg => #statMonitoring.bddData.dataValue[2]);
       Chars_TO_Strg(Chars := #statDataBuffer.rcv_bddResult,
                     pChars := 87,
                     Cnt := 8,
                     Strg => #statMonitoring.bddData.dataValue[3]);
       Chars_TO_Strg(Chars := #statDataBuffer.rcv_bddResult,
                     pChars := 111,
                     Cnt := 8,
                     Strg => #statMonitoring.bddData.dataValue[4]);
       Chars_TO_Strg(Chars := #statDataBuffer.rcv_bddResult,
                     pChars := 135,
                     Cnt := 8,
                     Strg => #statMonitoring.bddData.dataValue[5]);
       Chars_TO_Strg(Chars := #statDataBuffer.rcv_bddResult,
                     pChars := 159,
                     Cnt := 8,
                     Strg => #statMonitoring.bddData.dataValue[6]);
       Chars_TO_Strg(Chars := #statDataBuffer.rcv_bddResult,
                     pChars := 183,
                     Cnt := 8,
                     Strg => #statMonitoring.bddData.dataValue[7]);
       Chars_TO_Strg(Chars := #statDataBuffer.rcv_bddResult,
                     pChars := 207,
                     Cnt := 8,
                     Strg => #statMonitoring.bddData.dataValue[8]);
       Chars_TO_Strg(Chars := #statDataBuffer.rcv_bddResult,
                     pChars := 231,
                     Cnt := 8,
                     Strg => #statMonitoring.bddData.dataValue[9]);

       Chars_TO_Strg(Chars := #statDataBuffer.rcv_bddResult,
                     pChars := 255,
                     Cnt := 8,
                     Strg => #statMonitoring.bddData.dataValue[10]);
       Chars_TO_Strg(Chars := #statDataBuffer.rcv_bddResult,
                     pChars := 279,
                     Cnt := 8,
                     Strg => #statMonitoring.bddData.dataValue[11]);
       Chars_TO_Strg(Chars := #statDataBuffer.rcv_bddResult,
                     pChars := 303,
                     Cnt := 8,
                     Strg => #statMonitoring.bddData.dataValue[12]);
       Chars_TO_Strg(Chars := #statDataBuffer.rcv_bddResult,
                     pChars := 327,
                     Cnt := 8,
                     Strg => #statMonitoring.bddData.dataValue[13]);
       Chars_TO_Strg(Chars := #statDataBuffer.rcv_bddResult,
                     pChars := 351,
                     Cnt := 8,
                     Strg => #statMonitoring.bddData.dataValue[14]);
       Chars_TO_Strg(Chars := #statDataBuffer.rcv_bddResult,
                     pChars := 375,
                     Cnt := 8,
                     Strg => #statMonitoring.bddData.dataValue[15]);
       Chars_TO_Strg(Chars := #statDataBuffer.rcv_bddResult,
                     pChars := 399,
                     Cnt := 8,
                     Strg => #statMonitoring.bddData.dataValue[16]);
       Chars_TO_Strg(Chars := #statDataBuffer.rcv_bddResult,
                     pChars := 423,
                     Cnt := 8,
                     Strg => #statMonitoring.bddData.dataValue[17]);
       Chars_TO_Strg(Chars := #statDataBuffer.rcv_bddResult,
                     pChars := 447,
                     Cnt := 8,
                     Strg => #statMonitoring.bddData.dataValue[18]);
       Chars_TO_Strg(Chars := #statDataBuffer.rcv_bddResult,
                     pChars := 471,
                     Cnt := 8,
                     Strg => #statMonitoring.bddData.dataValue[19]);

       Chars_TO_Strg(Chars := #statDataBuffer.rcv_bddResult,
                     pChars := 495,
                     Cnt := 8,
                     Strg => #statMonitoring.bddData.dataValue[20]);
       Chars_TO_Strg(Chars := #statDataBuffer.rcv_bddResult,
                     pChars := 519,
                     Cnt := 8,
                     Strg => #statMonitoring.bddData.dataValue[21]);
       Chars_TO_Strg(Chars := #statDataBuffer.rcv_bddResult,
                     pChars := 543,
                     Cnt := 8,
                     Strg => #statMonitoring.bddData.dataValue[22]);
       Chars_TO_Strg(Chars := #statDataBuffer.rcv_bddResult,
                     pChars := 567,
                     Cnt := 8,
                     Strg => #statMonitoring.bddData.dataValue[23]);
       Chars_TO_Strg(Chars := #statDataBuffer.rcv_bddResult,
                     pChars := 591,
                     Cnt := 8,
                     Strg => #statMonitoring.bddData.dataValue[24]);
       Chars_TO_Strg(Chars := #statDataBuffer.rcv_bddResult,
                     pChars := 615,
                     Cnt := 8,
                     Strg => #statMonitoring.bddData.dataValue[25]);
       Chars_TO_Strg(Chars := #statDataBuffer.rcv_bddResult,
                     pChars := 639,
                     Cnt := 8,
                     Strg => #statMonitoring.bddData.dataValue[26]);
       Chars_TO_Strg(Chars := #statDataBuffer.rcv_bddResult,
                     pChars := 663,
                     Cnt := 8,
                     Strg => #statMonitoring.bddData.dataValue[27]);
       Chars_TO_Strg(Chars := #statDataBuffer.rcv_bddResult,
                     pChars := 687,
                     Cnt := 8,
                     Strg => #statMonitoring.bddData.dataValue[28]);
       Chars_TO_Strg(Chars := #statDataBuffer.rcv_bddResult,
                     pChars := 711,
                     Cnt := 8,
                     Strg => #statMonitoring.bddData.dataValue[29]);

       Chars_TO_Strg(Chars := #statDataBuffer.rcv_bddResult,
                     pChars := 735,
                     Cnt := 8,
                     Strg => #statMonitoring.bddData.dataValue[30]);
       Chars_TO_Strg(Chars := #statDataBuffer.rcv_bddResult,
                     pChars := 759,
                     Cnt := 8,
                     Strg => #statMonitoring.bddData.dataValue[31]);
       Chars_TO_Strg(Chars := #statDataBuffer.rcv_bddResult,
                     pChars := 783,
                     Cnt := 8,
                     Strg => #statMonitoring.bddData.dataValue[32]);
       Chars_TO_Strg(Chars := #statDataBuffer.rcv_bddResult,
                     pChars := 807,
                     Cnt := 8,
                     Strg => #statMonitoring.bddData.dataValue[33]);
       Chars_TO_Strg(Chars := #statDataBuffer.rcv_bddResult,
                     pChars := 831,
                     Cnt := 8,
                     Strg => #statMonitoring.bddData.dataValue[34]);
       Chars_TO_Strg(Chars := #statDataBuffer.rcv_bddResult,
                     pChars := 855,
                     Cnt := 8,
                     Strg => #statMonitoring.bddData.dataValue[35]);
       Chars_TO_Strg(Chars := #statDataBuffer.rcv_bddResult,
                     pChars := 879,
                     Cnt := 8,
                     Strg => #statMonitoring.bddData.dataValue[36]);
       Chars_TO_Strg(Chars := #statDataBuffer.rcv_bddResult,
                     pChars := 903,
                     Cnt := 8,
                     Strg => #statMonitoring.bddData.dataValue[37]);
       Chars_TO_Strg(Chars := #statDataBuffer.rcv_bddResult,
                     pChars := 927,
                     Cnt := 8,
                     Strg => #statMonitoring.bddData.dataValue[38]);
       Chars_TO_Strg(Chars := #statDataBuffer.rcv_bddResult,
                     pChars := 951,
                     Cnt := 8,
                     Strg => #statMonitoring.bddData.dataValue[39]);

       Chars_TO_Strg(Chars := #statDataBuffer.rcv_bddResult,
                     pChars := 975,
                     Cnt := 8,
                     Strg => #statMonitoring.bddData.dataValue[40]);
       Chars_TO_Strg(Chars := #statDataBuffer.rcv_bddResult,
                     pChars := 999,
                     Cnt := 8,
                     Strg => #statMonitoring.bddData.dataValue[41]);
       Chars_TO_Strg(Chars := #statDataBuffer.rcv_bddResult,
                     pChars := 1023,
                     Cnt := 8,
                     Strg => #statMonitoring.bddData.dataValue[42]);
       Chars_TO_Strg(Chars := #statDataBuffer.rcv_bddResult,
                     pChars := 1047,
                     Cnt := 8,
                     Strg => #statMonitoring.bddData.dataValue[43]);
       Chars_TO_Strg(Chars := #statDataBuffer.rcv_bddResult,
                     pChars := 1071,
                     Cnt := 8,
                     Strg => #statMonitoring.bddData.dataValue[44]);
       Chars_TO_Strg(Chars := #statDataBuffer.rcv_bddResult,
                     pChars := 1095,
                     Cnt := 8,
                     Strg => #statMonitoring.bddData.dataValue[45]);
       Chars_TO_Strg(Chars := #statDataBuffer.rcv_bddResult,
                     pChars := 1119,
                     Cnt := 8,
                     Strg => #statMonitoring.bddData.dataValue[46]);
       Chars_TO_Strg(Chars := #statDataBuffer.rcv_bddResult,
                     pChars := 1143,
                     Cnt := 8,
                     Strg => #statMonitoring.bddData.dataValue[47]);
       Chars_TO_Strg(Chars := #statDataBuffer.rcv_bddResult,
                     pChars := 1167,
                     Cnt := 8,
                     Strg => #statMonitoring.bddData.dataValue[48]);
       Chars_TO_Strg(Chars := #statDataBuffer.rcv_bddResult,
                     pChars := 1191,
                     Cnt := 8,
                     Strg => #statMonitoring.bddData.dataValue[49]);

       Chars_TO_Strg(Chars := #statDataBuffer.rcv_bddResult,
                     pChars := 1215,
                     Cnt := 8,
                     Strg => #statMonitoring.bddData.dataValue[50]);
       Chars_TO_Strg(Chars := #statDataBuffer.rcv_bddResult,
                     pChars := 1239,
                     Cnt := 8,
                     Strg => #statMonitoring.bddData.dataValue[51]);
       Chars_TO_Strg(Chars := #statDataBuffer.rcv_bddResult,
                     pChars := 1263,
                     Cnt := 8,
                     Strg => #statMonitoring.bddData.dataValue[52]);
       Chars_TO_Strg(Chars := #statDataBuffer.rcv_bddResult,
                     pChars := 1287,
                     Cnt := 8,
                     Strg => #statMonitoring.bddData.dataValue[53]);
       Chars_TO_Strg(Chars := #statDataBuffer.rcv_bddResult,
                     pChars := 1311,
                     Cnt := 8,
                     Strg => #statMonitoring.bddData.dataValue[54]);
       Chars_TO_Strg(Chars := #statDataBuffer.rcv_bddResult,
                     pChars := 1335,
                     Cnt := 8,
                     Strg => #statMonitoring.bddData.dataValue[55]);
       Chars_TO_Strg(Chars := #statDataBuffer.rcv_bddResult,
                     pChars := 1359,
                     Cnt := 8,
                     Strg => #statMonitoring.bddData.dataValue[56]);
       Chars_TO_Strg(Chars := #statDataBuffer.rcv_bddResult,
                     pChars := 1383,
                     Cnt := 8,
                     Strg => #statMonitoring.bddData.dataValue[57]);
       Chars_TO_Strg(Chars := #statDataBuffer.rcv_bddResult,
                     pChars := 1407,
                     Cnt := 8,
                     Strg => #statMonitoring.bddData.dataValue[58]);
       Chars_TO_Strg(Chars := #statDataBuffer.rcv_bddResult,
                     pChars := 1431,
                     Cnt := 8,
                     Strg => #statMonitoring.bddData.dataValue[59]);

       Chars_TO_Strg(Chars := #statDataBuffer.rcv_bddResult,
                     pChars := 1455,
                     Cnt := 8,
                     Strg => #statMonitoring.bddData.dataValue[60]);
       Chars_TO_Strg(Chars := #statDataBuffer.rcv_bddResult,
                     pChars := 1479,
                     Cnt := 8,
                     Strg => #statMonitoring.bddData.dataValue[61]);
       Chars_TO_Strg(Chars := #statDataBuffer.rcv_bddResult,
                     pChars := 1503,
                     Cnt := 8,
                     Strg => #statMonitoring.bddData.dataValue[62]);
       Chars_TO_Strg(Chars := #statDataBuffer.rcv_bddResult,
                     pChars := 1527,
                     Cnt := 8,
                     Strg => #statMonitoring.bddData.dataValue[63]);
       Chars_TO_Strg(Chars := #statDataBuffer.rcv_bddResult,
                     pChars := 1551,
                     Cnt := 8,
                     Strg => #statMonitoring.bddData.dataValue[64]);
       Chars_TO_Strg(Chars := #statDataBuffer.rcv_bddResult,
                     pChars := 1575,
                     Cnt := 8,
                     Strg => #statMonitoring.bddData.dataValue[65]);
       Chars_TO_Strg(Chars := #statDataBuffer.rcv_bddResult,
                     pChars := 1599,
                     Cnt := 8,
                     Strg => #statMonitoring.bddData.dataValue[66]);
       Chars_TO_Strg(Chars := #statDataBuffer.rcv_bddResult,
                     pChars := 1623,
                     Cnt := 8,
                     Strg => #statMonitoring.bddData.dataValue[67]);
       Chars_TO_Strg(Chars := #statDataBuffer.rcv_bddResult,
                     pChars := 1647,
                     Cnt := 8,
                     Strg => #statMonitoring.bddData.dataValue[68]);
       Chars_TO_Strg(Chars := #statDataBuffer.rcv_bddResult,
                     pChars := 1671,
                     Cnt := 8,
                     Strg => #statMonitoring.bddData.dataValue[69]);

       Chars_TO_Strg(Chars := #statDataBuffer.rcv_bddResult,
                     pChars := 1695,
                     Cnt := 8,
                     Strg => #statMonitoring.bddData.dataValue[70]);
       Chars_TO_Strg(Chars := #statDataBuffer.rcv_bddResult,
                     pChars := 1719,
                     Cnt := 8,
                     Strg => #statMonitoring.bddData.dataValue[71]);
       Chars_TO_Strg(Chars := #statDataBuffer.rcv_bddResult,
                     pChars := 1743,
                     Cnt := 8,
                     Strg => #statMonitoring.bddData.dataValue[72]);
       Chars_TO_Strg(Chars := #statDataBuffer.rcv_bddResult,
                     pChars := 1767,
                     Cnt := 8,
                     Strg => #statMonitoring.bddData.dataValue[73]);
       Chars_TO_Strg(Chars := #statDataBuffer.rcv_bddResult,
                     pChars := 1791,
                     Cnt := 8,
                     Strg => #statMonitoring.bddData.dataValue[74]);
       Chars_TO_Strg(Chars := #statDataBuffer.rcv_bddResult,
                     pChars := 1815,
                     Cnt := 8,
                     Strg => #statMonitoring.bddData.dataValue[75]);
       Chars_TO_Strg(Chars := #statDataBuffer.rcv_bddResult,
                     pChars := 1839,
                     Cnt := 8,
                     Strg => #statMonitoring.bddData.dataValue[76]);
       Chars_TO_Strg(Chars := #statDataBuffer.rcv_bddResult,
                     pChars := 1863,
                     Cnt := 8,
                     Strg => #statMonitoring.bddData.dataValue[77]);
       Chars_TO_Strg(Chars := #statDataBuffer.rcv_bddResult,
                     pChars := 1887,
                     Cnt := 8,
                     Strg => #statMonitoring.bddData.dataValue[78]);
       Chars_TO_Strg(Chars := #statDataBuffer.rcv_bddResult,
                     pChars := 1911,
                     Cnt := 8,
                     Strg => #statMonitoring.bddData.dataValue[79]);

       Chars_TO_Strg(Chars := #statDataBuffer.rcv_bddResult,
                     pChars := 1935,
                     Cnt := 8,
                     Strg => #statMonitoring.bddData.dataValue[80]);
       Chars_TO_Strg(Chars := #statDataBuffer.rcv_bddResult,
                     pChars := 1959,
                     Cnt := 8,
                     Strg => #statMonitoring.bddData.dataValue[81]);
       Chars_TO_Strg(Chars := #statDataBuffer.rcv_bddResult,
                     pChars := 1983,
                     Cnt := 8,
                     Strg => #statMonitoring.bddData.dataValue[82]);
       Chars_TO_Strg(Chars := #statDataBuffer.rcv_bddResult,
                     pChars := 2007,
                     Cnt := 8,
                     Strg => #statMonitoring.bddData.dataValue[83]);
       Chars_TO_Strg(Chars := #statDataBuffer.rcv_bddResult,
                     pChars := 2031,
                     Cnt := 8,
                     Strg => #statMonitoring.bddData.dataValue[84]);
       Chars_TO_Strg(Chars := #statDataBuffer.rcv_bddResult,
                     pChars := 2055,
                     Cnt := 8,
                     Strg => #statMonitoring.bddData.dataValue[85]);
       Chars_TO_Strg(Chars := #statDataBuffer.rcv_bddResult,
                     pChars := 2079,
                     Cnt := 8,
                     Strg => #statMonitoring.bddData.dataValue[86]);
       Chars_TO_Strg(Chars := #statDataBuffer.rcv_bddResult,
                     pChars := 2103,
                     Cnt := 8,
                     Strg => #statMonitoring.bddData.dataValue[87]);
       Chars_TO_Strg(Chars := #statDataBuffer.rcv_bddResult,
                     pChars := 2127,
                     Cnt := 8,
                     Strg => #statMonitoring.bddData.dataValue[88]);
       Chars_TO_Strg(Chars := #statDataBuffer.rcv_bddResult,
                     pChars := 2151,
                     Cnt := 8,
                     Strg => #statMonitoring.bddData.dataValue[89]);

